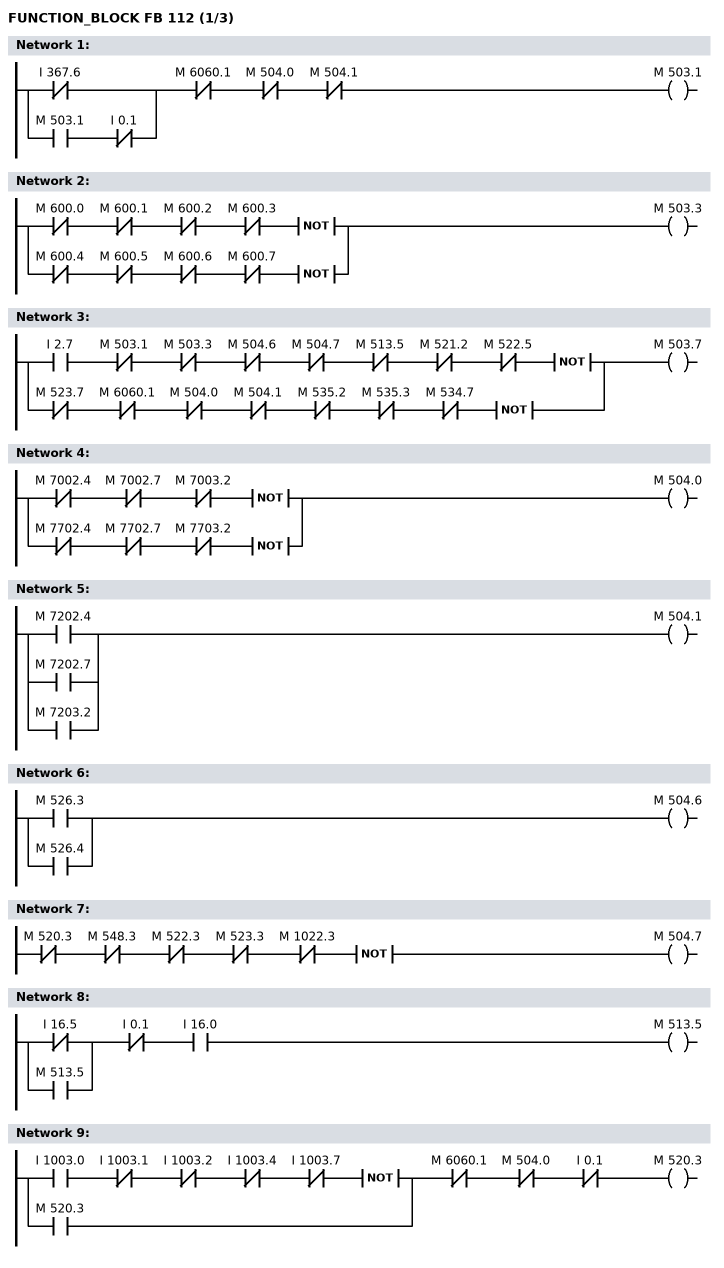

      A(    ;
      ON    I    367.6;
      O     ;
      A     M    503.1;
      AN    I      0.1;
      )     ;
      AN    M   6060.1;
      AN    M    504.0;
      AN    M    504.1;
      =     M    503.1;
NETWORK
TITLE =

      AN    M    600.0;
      AN    M    600.1;
      AN    M    600.2;
      AN    M    600.3;
      NOT   ;
      O(    ;
      AN    M    600.4;
      AN    M    600.5;
      AN    M    600.6;
      AN    M    600.7;
      NOT   ;
      )     ;
      =     M    503.3;
NETWORK
TITLE =

      A     I      2.7;
      AN    M    503.1;
      AN    M    503.3;
      AN    M    504.6;
      AN    M    504.7;
      AN    M    513.5;
      AN    M    521.2;
      AN    M    522.5;
      NOT   ;
      O(    ;
      AN    M    523.7;
      AN    M   6060.1;
      AN    M    504.0;
      AN    M    504.1;
      AN    M    535.2;
      AN    M    535.3;
      AN    M    534.7;
      NOT   ;
      )     ;
      =     M    503.7;
NETWORK
TITLE =

      AN    M   7002.4;
      AN    M   7002.7;
      AN    M   7003.2;
      NOT   ;
      O(    ;
      AN    M   7702.4;
      AN    M   7702.7;
      AN    M   7703.2;
      NOT   ;
      )     ;
      =     M    504.0;
NETWORK
TITLE =

      O     M   7202.4;
      O     M   7202.7;
      O     M   7203.2;
      =     M    504.1;
NETWORK
TITLE =

      O     M    526.3;
      O     M    526.4;
      =     M    504.6;
NETWORK
TITLE =

      AN    M    520.3;
      AN    M    548.3;
      AN    M    522.3;
      AN    M    523.3;
      AN    M   1022.3;
      NOT   ;
      =     M    504.7;
NETWORK
TITLE =

      A(    ;
      ON    I     16.5;
      O     M    513.5;
      )     ;
      AN    I      0.1;
      A     I     16.0;
      =     M    513.5;
NETWORK
TITLE =

      A(    ;
      A     I   1003.0;
      AN    I   1003.1;
      AN    I   1003.2;
      AN    I   1003.4;
      AN    I   1003.7;
      NOT   ;
      O     M    520.3;
      )     ;
      AN    M   6060.1;
      AN    M    504.0;
      AN    I      0.1;
      =     M    520.3;
NETWORK
TITLE =
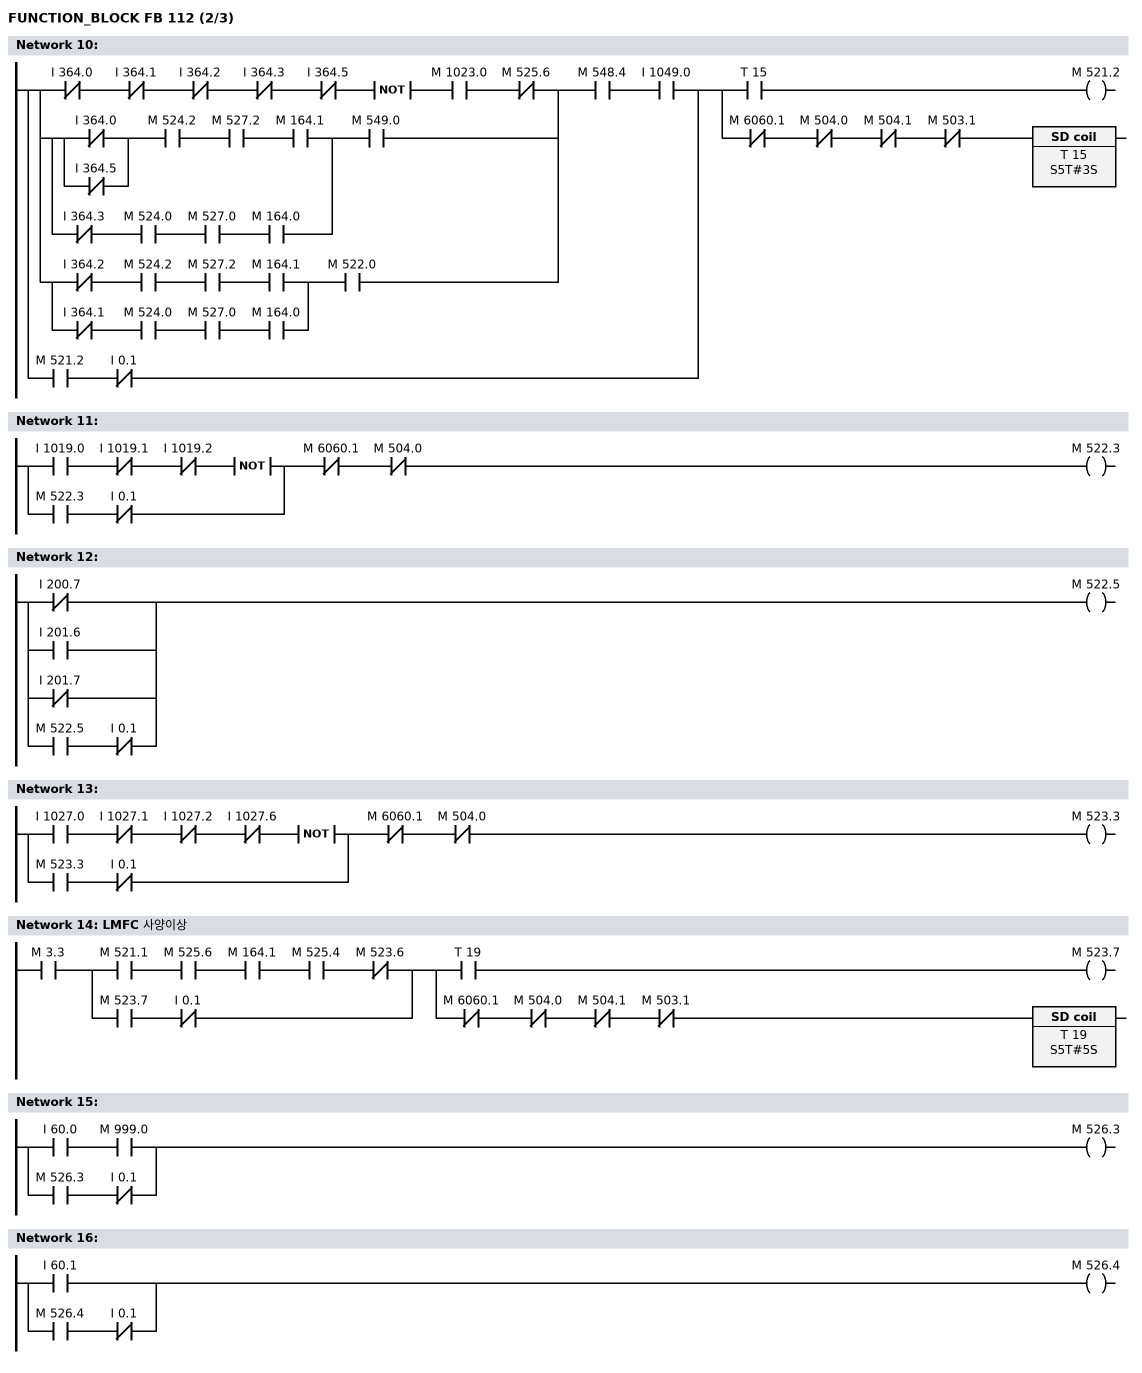

      A(    ;
      AN    I    364.0;
      AN    I    364.1;
      AN    I    364.2;
      AN    I    364.3;
      AN    I    364.5;
      NOT   ;
      A     M   1023.0;
      AN    M    525.6;
      O     ;
      A(    ;
      A(    ;
      ON    I    364.0;
      ON    I    364.5;
      )     ;
      A     M    524.2;
      A     M    527.2;
      A     M    164.1;
      O     ;
      AN    I    364.3;
      A     M    524.0;
      A     M    527.0;
      A     M    164.0;
      )     ;
      A     M    549.0;
      O     ;
      A(    ;
      AN    I    364.2;
      A     M    524.2;
      A     M    527.2;
      A     M    164.1;
      O     ;
      AN    I    364.1;
      A     M    524.0;
      A     M    527.0;
      A     M    164.0;
      )     ;
      A     M    522.0;
      )     ;
      A     M    548.4;
      A     I   1049.0;
      O     ;
      A     M    521.2;
      AN    I      0.1;
      =     L      0.0;
      A     L      0.0;
      A     T     15;
      =     M    521.2;
      A     L      0.0;
      AN    M   6060.1;
      AN    M    504.0;
      AN    M    504.1;
      AN    M    503.1;
      L     S5T#3S;
      SD    T     15;
NETWORK
TITLE =

      A(    ;
      A     I   1019.0;
      AN    I   1019.1;
      AN    I   1019.2;
      NOT   ;
      O     ;
      A     M    522.3;
      AN    I      0.1;
      )     ;
      AN    M   6060.1;
      AN    M    504.0;
      =     M    522.3;
NETWORK
TITLE =

      ON    I    200.7;
      O     I    201.6;
      ON    I    201.7;
      O     ;
      A     M    522.5;
      AN    I      0.1;
      =     M    522.5;
NETWORK
TITLE =

      A(    ;
      A     I   1027.0;
      AN    I   1027.1;
      AN    I   1027.2;
      AN    I   1027.6;
      NOT   ;
      O     ;
      A     M    523.3;
      AN    I      0.1;
      )     ;
      AN    M   6060.1;
      AN    M    504.0;
      =     M    523.3;
NETWORK
TITLE =LMFC 사양이상

      A     M      3.3;
      A(    ;
      A     M    521.1;
      A     M    525.6;
      A     M    164.1;
      A     M    525.4;
      AN    M    523.6;
      O     ;
      A     M    523.7;
      AN    I      0.1;
      )     ;
      =     L      0.0;
      A     L      0.0;
      A     T     19;
      =     M    523.7;
      A     L      0.0;
      AN    M   6060.1;
      AN    M    504.0;
      AN    M    504.1;
      AN    M    503.1;
      L     S5T#5S;
      SD    T     19;
NETWORK
TITLE =

      A     I     60.0;
      A     M    999.0;
      O     ;
      A     M    526.3;
      AN    I      0.1;
      =     M    526.3;
NETWORK
TITLE =

      O     I     60.1;
      O     ;
      A     M    526.4;
      AN    I      0.1;
      =     M    526.4;
NETWORK
TITLE =
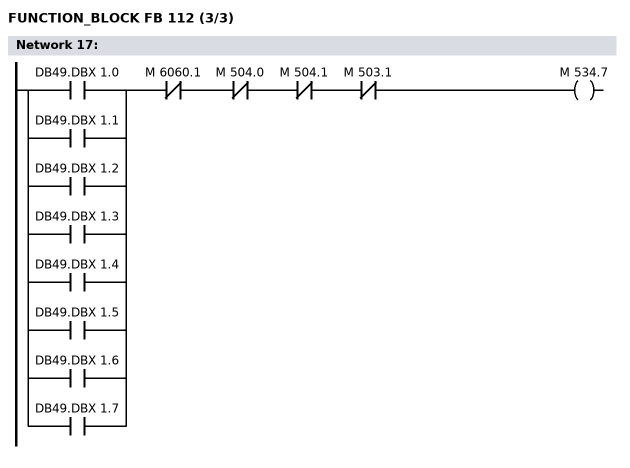

      A(    ;
      O     DB49.DBX    1.0;
      O     DB49.DBX    1.1;
      O     DB49.DBX    1.2;
      O     DB49.DBX    1.3;
      O     DB49.DBX    1.4;
      O     DB49.DBX    1.5;
      O     DB49.DBX    1.6;
      O     DB49.DBX    1.7;
      )     ;
      AN    M   6060.1;
      AN    M    504.0;
      AN    M    504.1;
      AN    M    503.1;
      =     M    534.7;
NETWORK
TITLE =

      A     M      3.3;
      =     L      0.0;
      A     L      0.0;
      A(    ;
      A     M    535.6;
      A(    ;
      ON    M    535.4;
      O     ;
      A     M    535.4;
      A(    ;
      A     I    367.1;
      A     I    367.3;
      O     ;
      AN    I    367.1;
      AN    I    367.3;
      O     ;
      A     M    124.0;
      A     I    367.1;
      AN    I    367.3;
      O     ;
      A     M    124.1;
      AN    I    367.1;
      A     I    367.3;
      )     ;
      )     ;
      A     I   1009.1;
      O     ;
      A     M    535.2;
      AN    I      0.1;
      )     ;
      =     L      0.1;
      A     L      0.1;
      A     T     12;
      =     M    535.2;
      A     L      0.1;
      AN    M   6060.1;
      AN    M    504.0;
      AN    M    504.1;
      AN    M    503.1;
      L     S5T#1S;
      SD    T     12;
      A     L      0.0;
      A(    ;
      A     M    535.7;
      AN    M    535.5;
      A     I   1002.2;
      O     ;
      A     M    535.3;
      AN    I      0.1;
      )     ;
      =     L      0.1;
      A     L      0.1;
      A     T     13;
      =     M    535.3;
      A     L      0.1;
      AN    M   6060.1;
      AN    M    504.0;
      AN    M    504.1;
      AN    M    503.1;
      L     S5T#1S;
      SD    T     13;
NETWORK
TITLE =
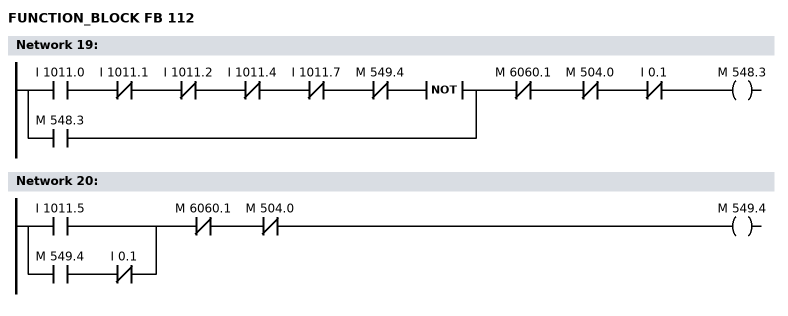

      A(    ;
      A     I   1011.0;
      AN    I   1011.1;
      AN    I   1011.2;
      AN    I   1011.4;
      AN    I   1011.7;
      AN    M    549.4;
      NOT   ;
      O     M    548.3;
      )     ;
      AN    M   6060.1;
      AN    M    504.0;
      AN    I      0.1;
      =     M    548.3;
NETWORK
TITLE =

      A(    ;
      O     I   1011.5;
      O     ;
      A     M    549.4;
      AN    I      0.1;
      )     ;
      AN    M   6060.1;
      AN    M    504.0;
      =     M    549.4;
END_FUNCTION_BLOCK

DATA_BLOCK DB 112
TITLE =
VERSION : 0.0

 FB 112
BEGIN
END_DATA_BLOCK

FUNCTION FC 112 : VOID
TITLE =
VERSION : 0.1

BEGIN
NETWORK
TITLE =

      AN    OV;
      =     L      0.0;
      A     L      0.0;
      A     I    364.6;
      AN    I    364.7;
      A     I    365.0;
      AN    I    365.1;
      =     M    524.0;
      A     L      0.0;
      AN    I    364.6;
      A     I    364.7;
      AN    I    365.0;
      A     I    365.1;
      =     M    524.1;
NETWORK
TITLE =

      AN    OV;
      =     L      0.0;
      A     L      0.0;
      A     I    365.2;
      AN    I    365.3;
      A     I    365.4;
      AN    I    365.5;
      =     M    524.2;
      A     L      0.0;
      AN    I    365.2;
      A     I    365.3;
      AN    I    365.4;
      A     I    365.5;
      =     M    524.3;
NETWORK
TITLE =

      AN    OV;
      =     L      0.0;
      A     L      0.0;
      A     I    366.0;
      AN    I    366.1;
      A     I    366.2;
      AN    I    366.3;
      =     M    527.0;
      A     L      0.0;
      AN    I    366.0;
      A     I    366.1;
      AN    I    366.2;
      A     I    366.3;
      =     M    527.1;
NETWORK
TITLE =

      AN    OV;
      =     L      0.0;
      A     L      0.0;
      A     I    366.4;
      AN    I    366.5;
      A     I    366.6;
      AN    I    366.7;
      =     M    527.2;
      A     L      0.0;
      AN    I    366.4;
      A     I    366.5;
      AN    I    366.6;
      A     I    366.7;
      =     M    527.3;
NETWORK
TITLE =
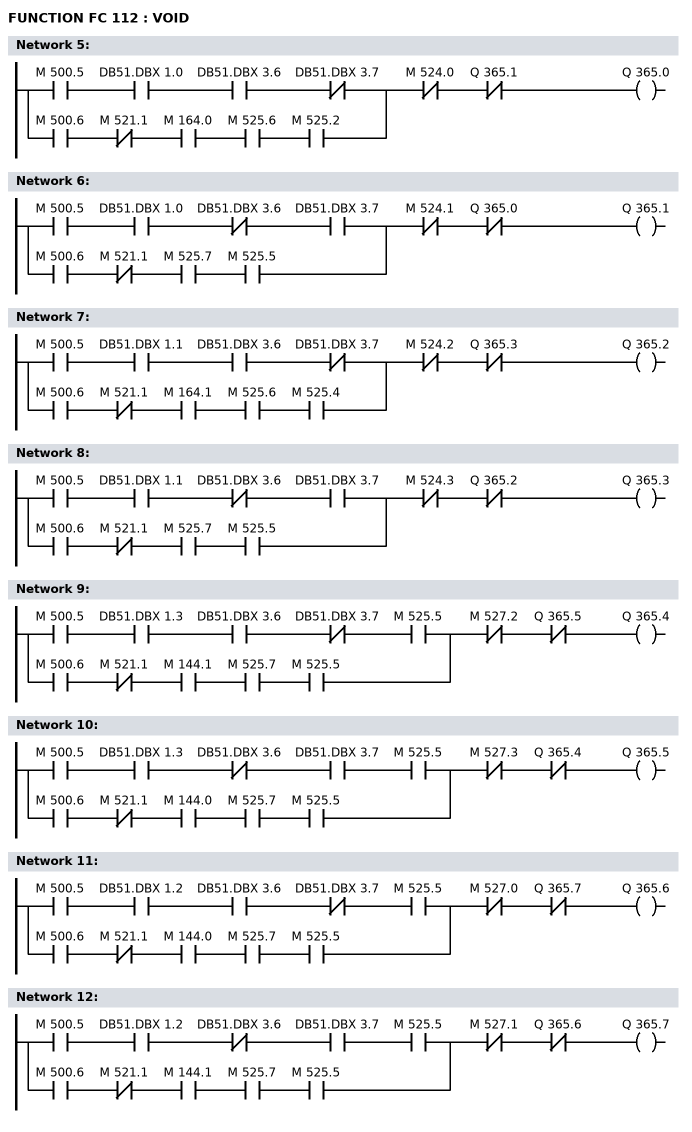

      A(    ;
      A     M    500.5;
      A     DB51.DBX    1.0;
      A     DB51.DBX    3.6;
      AN    DB51.DBX    3.7;
      O     ;
      A     M    500.6;
      AN    M    521.1;
      A     M    164.0;
      A     M    525.6;
      A     M    525.2;
      )     ;
      AN    M    524.0;
      AN    Q    365.1;
      =     Q    365.0;
NETWORK
TITLE =

      A(    ;
      A     M    500.5;
      A     DB51.DBX    1.0;
      AN    DB51.DBX    3.6;
      A     DB51.DBX    3.7;
      O     ;
      A     M    500.6;
      AN    M    521.1;
      A     M    525.7;
      A     M    525.5;
      )     ;
      AN    M    524.1;
      AN    Q    365.0;
      =     Q    365.1;
NETWORK
TITLE =

      A(    ;
      A     M    500.5;
      A     DB51.DBX    1.1;
      A     DB51.DBX    3.6;
      AN    DB51.DBX    3.7;
      O     ;
      A     M    500.6;
      AN    M    521.1;
      A     M    164.1;
      A     M    525.6;
      A     M    525.4;
      )     ;
      AN    M    524.2;
      AN    Q    365.3;
      =     Q    365.2;
NETWORK
TITLE =

      A(    ;
      A     M    500.5;
      A     DB51.DBX    1.1;
      AN    DB51.DBX    3.6;
      A     DB51.DBX    3.7;
      O     ;
      A     M    500.6;
      AN    M    521.1;
      A     M    525.7;
      A     M    525.5;
      )     ;
      AN    M    524.3;
      AN    Q    365.2;
      =     Q    365.3;
NETWORK
TITLE =

      A(    ;
      A     M    500.5;
      A     DB51.DBX    1.3;
      A     DB51.DBX    3.6;
      AN    DB51.DBX    3.7;
      A     M    525.5;
      O     ;
      A     M    500.6;
      AN    M    521.1;
      A     M    144.1;
      A     M    525.7;
      A     M    525.5;
      )     ;
      AN    M    527.2;
      AN    Q    365.5;
      =     Q    365.4;
NETWORK
TITLE =

      A(    ;
      A     M    500.5;
      A     DB51.DBX    1.3;
      AN    DB51.DBX    3.6;
      A     DB51.DBX    3.7;
      A     M    525.5;
      O     ;
      A     M    500.6;
      AN    M    521.1;
      A     M    144.0;
      A     M    525.7;
      A     M    525.5;
      )     ;
      AN    M    527.3;
      AN    Q    365.4;
      =     Q    365.5;
NETWORK
TITLE =

      A(    ;
      A     M    500.5;
      A     DB51.DBX    1.2;
      A     DB51.DBX    3.6;
      AN    DB51.DBX    3.7;
      A     M    525.5;
      O     ;
      A     M    500.6;
      AN    M    521.1;
      A     M    144.0;
      A     M    525.7;
      A     M    525.5;
      )     ;
      AN    M    527.0;
      AN    Q    365.7;
      =     Q    365.6;
NETWORK
TITLE =

      A(    ;
      A     M    500.5;
      A     DB51.DBX    1.2;
      AN    DB51.DBX    3.6;
      A     DB51.DBX    3.7;
      A     M    525.5;
      O     ;
      A     M    500.6;
      AN    M    521.1;
      A     M    144.1;
      A     M    525.7;
      A     M    525.5;
      )     ;
      AN    M    527.1;
      AN    Q    365.6;
      =     Q    365.7;
END_FUNCTION

FUNCTION FC 113 : VOID
TITLE =
VERSION : 0.1

BEGIN
NETWORK
TITLE =

      A     I   1000.0;
      JNB   _001;
      L     0;
      T     MW   590;
_001: NOP   0;
NETWORK
TITLE =

      AN    OV;
      =     L      0.0;
      A     L      0.0;
      A     M    104.1;
      =     L      0.1;
      A     L      0.1;
      A     T    363;
      A(    ;
      L     1;
      L     DB59.DBW   34;
      ==I   ;
      )     ;
      A(    ;
      L     1;
      L     DB59.DBW   30;
      ==I   ;
      )     ;
      A     M    550.3;
      JNB   _002;
      L     23;
      T     MB   591;
_002: NOP   0;
      A     L      0.1;
      A     T    364;
      A(    ;
      L     1;
      L     DB59.DBW   44;
      ==I   ;
      )     ;
      A(    ;
      L     1;
      L     DB59.DBW   40;
      ==I   ;
      )     ;
      A     M    550.4;
      JNB   _003;
      L     24;
      T     MB   591;
_003: NOP   0;
      A     L      0.1;
      A     T    365;
      A(    ;
      L     1;
      L     DB59.DBW   54;
      ==I   ;
      )     ;
      A(    ;
      L     1;
      L     DB59.DBW   50;
      ==I   ;
      )     ;
      A     M    550.5;
      JNB   _004;
      L     25;
      T     MB   591;
_004: NOP   0;
      A     L      0.1;
      A     T    366;
      A(    ;
      L     1;
      L     DB59.DBW   64;
      ==I   ;
      )     ;
      A(    ;
      L     1;
      L     DB59.DBW   60;
      ==I   ;
      )     ;
      A     M    550.6;
      JNB   _005;
      L     26;
      T     MB   591;
_005: NOP   0;
      A     L      0.0;
      A     M    104.0;
      =     L      0.1;
      A     L      0.1;
      A     T    363;
      A(    ;
      L     1;
      L     DB59.DBW   34;
      ==I   ;
      )     ;
      A(    ;
      L     2;
      L     DB59.DBW   30;
      ==I   ;
      )     ;
      A     M    554.3;
      JNB   _006;
      L     3;
      T     MB   591;
_006: NOP   0;
      A     L      0.1;
      A     T    364;
      A(    ;
      L     1;
      L     DB59.DBW   44;
      ==I   ;
      )     ;
      A(    ;
      L     2;
      L     DB59.DBW   40;
      ==I   ;
      )     ;
      A     M    554.4;
      JNB   _007;
      L     4;
      T     MB   591;
_007: NOP   0;
      A     L      0.1;
      A     T    365;
      A(    ;
      L     1;
      L     DB59.DBW   54;
      ==I   ;
      )     ;
      A(    ;
      L     2;
      L     DB59.DBW   50;
      ==I   ;
      )     ;
      A     M    554.5;
      JNB   _008;
      L     5;
      T     MB   591;
_008: NOP   0;
      A     L      0.1;
      A     T    366;
      A(    ;
      L     1;
      L     DB59.DBW   64;
      ==I   ;
      )     ;
      A(    ;
      L     2;
      L     DB59.DBW   60;
      ==I   ;
      )     ;
      A     M    554.6;
      JNB   _009;
      L     6;
      T     MB   591;
_009: NOP   0;
NETWORK
TITLE =

      AN    OV;
      =     L      0.0;
      A     L      0.0;
      A     M    104.1;
      =     L      0.1;
      A     L      0.1;
      A     T    369;
      A(    ;
      L     1;
      L     DB59.DBW   94;
      ==I   ;
      )     ;
      A(    ;
      L     1;
      L     DB59.DBW   90;
      ==I   ;
      )     ;
      A     M    551.1;
      JNB   _00a;
      L     29;
      T     MB   591;
_00a: NOP   0;
      A     L      0.1;
      A     T    370;
      A(    ;
      L     1;
      L     DB59.DBW  104;
      ==I   ;
      )     ;
      A(    ;
      L     1;
      L     DB59.DBW  100;
      ==I   ;
      )     ;
      A     M    551.2;
      JNB   _00b;
      L     30;
      T     MB   591;
_00b: NOP   0;
      A     L      0.1;
      A     T    371;
      A(    ;
      L     1;
      L     DB59.DBW  114;
      ==I   ;
      )     ;
      A(    ;
      L     1;
      L     DB59.DBW  110;
      ==I   ;
      )     ;
      A     M    551.3;
      JNB   _00c;
      L     31;
      T     MB   591;
_00c: NOP   0;
      A     L      0.1;
      A     T    372;
      A(    ;
      L     1;
      L     DB59.DBW  124;
      ==I   ;
      )     ;
      A(    ;
      L     1;
      L     DB59.DBW  120;
      ==I   ;
      )     ;
      A     M    551.4;
      JNB   _00d;
      L     32;
      T     MB   591;
_00d: NOP   0;
      A     L      0.0;
      A     M    104.0;
      =     L      0.1;
      A     L      0.1;
      A     T    369;
      A(    ;
      L     1;
      L     DB59.DBW   94;
      ==I   ;
      )     ;
      A(    ;
      L     2;
      L     DB59.DBW   90;
      ==I   ;
      )     ;
      A     M    555.1;
      JNB   _00e;
      L     9;
      T     MB   591;
_00e: NOP   0;
      A     L      0.1;
      A     T    370;
      A(    ;
      L     1;
      L     DB59.DBW  104;
      ==I   ;
      )     ;
      A(    ;
      L     2;
      L     DB59.DBW  100;
      ==I   ;
      )     ;
      A     M    555.2;
      JNB   _00f;
      L     10;
      T     MB   591;
_00f: NOP   0;
      A     L      0.1;
      A     T    371;
      A(    ;
      L     1;
      L     DB59.DBW  114;
      ==I   ;
      )     ;
      A(    ;
      L     2;
      L     DB59.DBW  110;
      ==I   ;
      )     ;
      A     M    555.3;
      JNB   _010;
      L     11;
      T     MB   591;
_010: NOP   0;
      A     L      0.1;
      A     T    372;
      A(    ;
      L     1;
      L     DB59.DBW  124;
      ==I   ;
      )     ;
      A(    ;
      L     2;
      L     DB59.DBW  120;
      ==I   ;
      )     ;
      A     M    555.4;
      JNB   _011;
      L     12;
      T     MB   591;
_011: NOP   0;
NETWORK
TITLE =
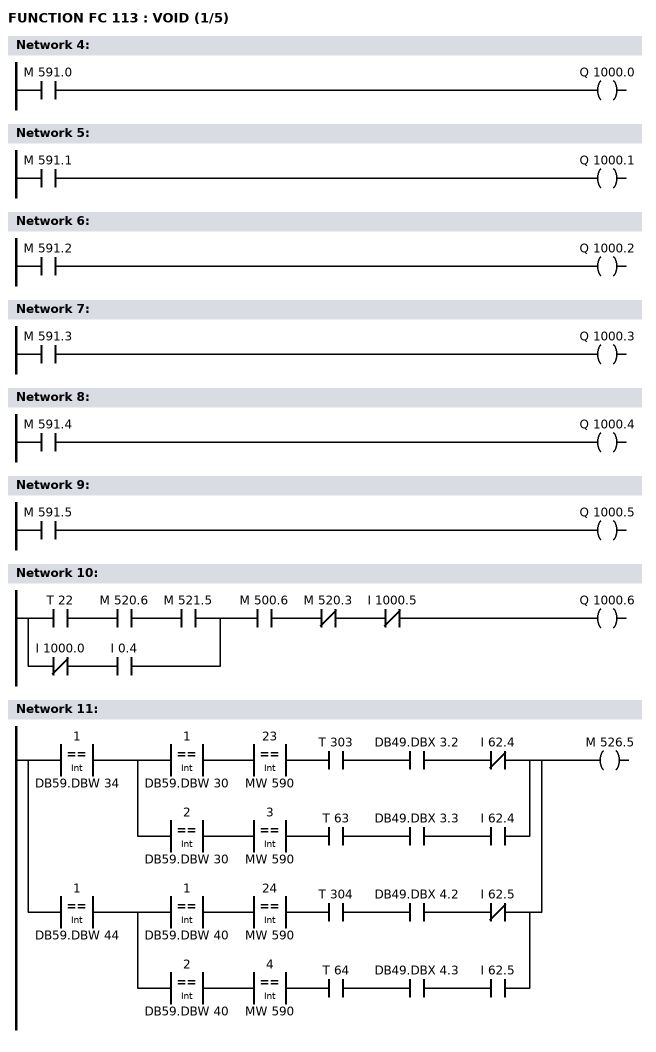

      A     M    591.0;
      =     Q   1000.0;
NETWORK
TITLE =

      A     M    591.1;
      =     Q   1000.1;
NETWORK
TITLE =

      A     M    591.2;
      =     Q   1000.2;
NETWORK
TITLE =

      A     M    591.3;
      =     Q   1000.3;
NETWORK
TITLE =

      A     M    591.4;
      =     Q   1000.4;
NETWORK
TITLE =

      A     M    591.5;
      =     Q   1000.5;
NETWORK
TITLE =

      A(    ;
      A     T     22;
      A     M    520.6;
      A     M    521.5;
      O     ;
      AN    I   1000.0;
      A     I      0.4;
      )     ;
      A     M    500.6;
      AN    M    520.3;
      AN    I   1000.5;
      =     Q   1000.6;
NETWORK
TITLE =

      A(    ;
      L     1;
      L     DB59.DBW   34;
      ==I   ;
      )     ;
      A(    ;
      A(    ;
      L     1;
      L     DB59.DBW   30;
      ==I   ;
      )     ;
      A(    ;
      L     23;
      L     MW   590;
      ==I   ;
      )     ;
      A     T    303;
      A     DB49.DBX    3.2;
      AN    I     62.4;
      O     ;
      A(    ;
      L     2;
      L     DB59.DBW   30;
      ==I   ;
      )     ;
      A(    ;
      L     3;
      L     MW   590;
      ==I   ;
      )     ;
      A     T     63;
      A     DB49.DBX    3.3;
      A     I     62.4;
      )     ;
      O     ;
      A(    ;
      L     1;
      L     DB59.DBW   44;
      ==I   ;
      )     ;
      A(    ;
      A(    ;
      L     1;
      L     DB59.DBW   40;
      ==I   ;
      )     ;
      A(    ;
      L     24;
      L     MW   590;
      ==I   ;
      )     ;
      A     T    304;
      A     DB49.DBX    4.2;
      AN    I     62.5;
      O     ;
      A(    ;
      L     2;
      L     DB59.DBW   40;
      ==I   ;
      )     ;
      A(    ;
      L     4;
      L     MW   590;
      ==I   ;
      )     ;
      A     T     64;
      A     DB49.DBX    4.3;
      A     I     62.5;
      )     ;
      =     M    526.5;
NETWORK
TITLE =
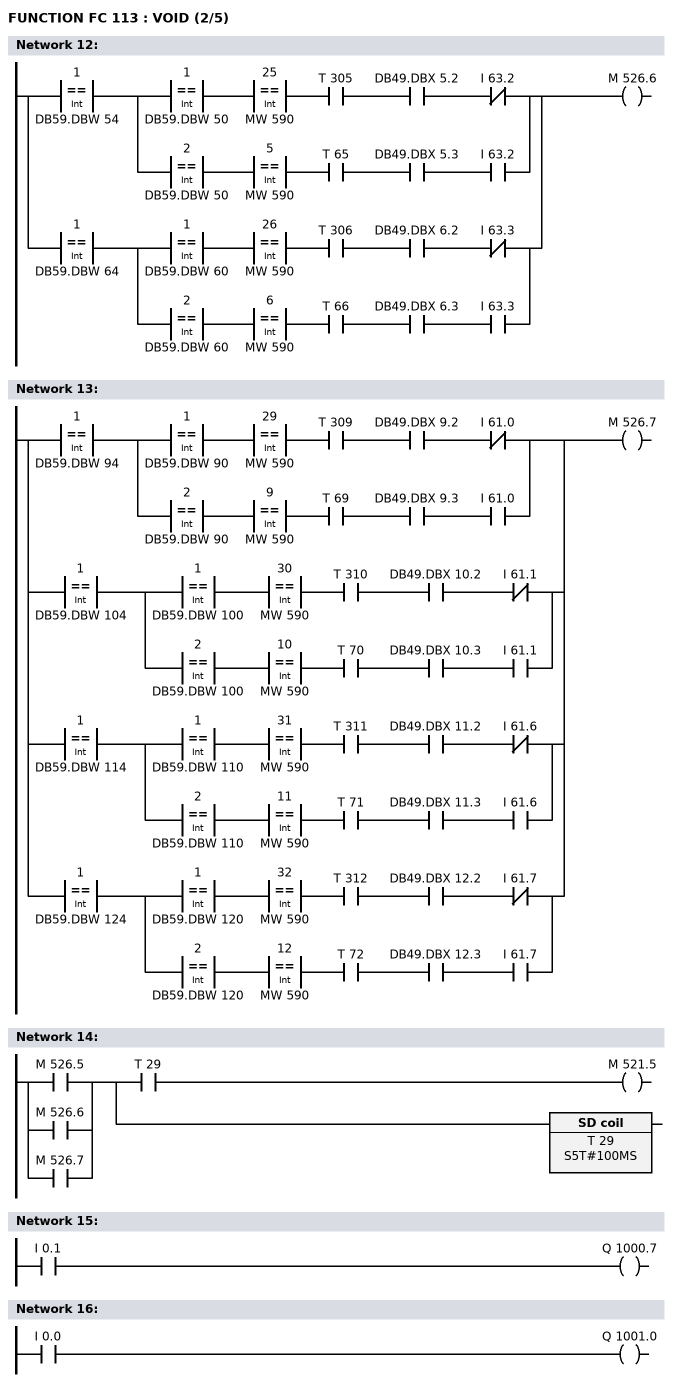

      A(    ;
      L     1;
      L     DB59.DBW   54;
      ==I   ;
      )     ;
      A(    ;
      A(    ;
      L     1;
      L     DB59.DBW   50;
      ==I   ;
      )     ;
      A(    ;
      L     25;
      L     MW   590;
      ==I   ;
      )     ;
      A     T    305;
      A     DB49.DBX    5.2;
      AN    I     63.2;
      O     ;
      A(    ;
      L     2;
      L     DB59.DBW   50;
      ==I   ;
      )     ;
      A(    ;
      L     5;
      L     MW   590;
      ==I   ;
      )     ;
      A     T     65;
      A     DB49.DBX    5.3;
      A     I     63.2;
      )     ;
      O     ;
      A(    ;
      L     1;
      L     DB59.DBW   64;
      ==I   ;
      )     ;
      A(    ;
      A(    ;
      L     1;
      L     DB59.DBW   60;
      ==I   ;
      )     ;
      A(    ;
      L     26;
      L     MW   590;
      ==I   ;
      )     ;
      A     T    306;
      A     DB49.DBX    6.2;
      AN    I     63.3;
      O     ;
      A(    ;
      L     2;
      L     DB59.DBW   60;
      ==I   ;
      )     ;
      A(    ;
      L     6;
      L     MW   590;
      ==I   ;
      )     ;
      A     T     66;
      A     DB49.DBX    6.3;
      A     I     63.3;
      )     ;
      =     M    526.6;
NETWORK
TITLE =

      A(    ;
      L     1;
      L     DB59.DBW   94;
      ==I   ;
      )     ;
      A(    ;
      A(    ;
      L     1;
      L     DB59.DBW   90;
      ==I   ;
      )     ;
      A(    ;
      L     29;
      L     MW   590;
      ==I   ;
      )     ;
      A     T    309;
      A     DB49.DBX    9.2;
      AN    I     61.0;
      O     ;
      A(    ;
      L     2;
      L     DB59.DBW   90;
      ==I   ;
      )     ;
      A(    ;
      L     9;
      L     MW   590;
      ==I   ;
      )     ;
      A     T     69;
      A     DB49.DBX    9.3;
      A     I     61.0;
      )     ;
      O     ;
      A(    ;
      L     1;
      L     DB59.DBW  104;
      ==I   ;
      )     ;
      A(    ;
      A(    ;
      L     1;
      L     DB59.DBW  100;
      ==I   ;
      )     ;
      A(    ;
      L     30;
      L     MW   590;
      ==I   ;
      )     ;
      A     T    310;
      A     DB49.DBX   10.2;
      AN    I     61.1;
      O     ;
      A(    ;
      L     2;
      L     DB59.DBW  100;
      ==I   ;
      )     ;
      A(    ;
      L     10;
      L     MW   590;
      ==I   ;
      )     ;
      A     T     70;
      A     DB49.DBX   10.3;
      A     I     61.1;
      )     ;
      O     ;
      A(    ;
      L     1;
      L     DB59.DBW  114;
      ==I   ;
      )     ;
      A(    ;
      A(    ;
      L     1;
      L     DB59.DBW  110;
      ==I   ;
      )     ;
      A(    ;
      L     31;
      L     MW   590;
      ==I   ;
      )     ;
      A     T    311;
      A     DB49.DBX   11.2;
      AN    I     61.6;
      O     ;
      A(    ;
      L     2;
      L     DB59.DBW  110;
      ==I   ;
      )     ;
      A(    ;
      L     11;
      L     MW   590;
      ==I   ;
      )     ;
      A     T     71;
      A     DB49.DBX   11.3;
      A     I     61.6;
      )     ;
      O     ;
      A(    ;
      L     1;
      L     DB59.DBW  124;
      ==I   ;
      )     ;
      A(    ;
      A(    ;
      L     1;
      L     DB59.DBW  120;
      ==I   ;
      )     ;
      A(    ;
      L     32;
      L     MW   590;
      ==I   ;
      )     ;
      A     T    312;
      A     DB49.DBX   12.2;
      AN    I     61.7;
      O     ;
      A(    ;
      L     2;
      L     DB59.DBW  120;
      ==I   ;
      )     ;
      A(    ;
      L     12;
      L     MW   590;
      ==I   ;
      )     ;
      A     T     72;
      A     DB49.DBX   12.3;
      A     I     61.7;
      )     ;
      =     M    526.7;
NETWORK
TITLE =

      O     M    526.5;
      O     M    526.6;
      O     M    526.7;
      =     L      0.0;
      A     L      0.0;
      A     T     29;
      =     M    521.5;
      A     L      0.0;
      BLD   102;
      L     S5T#100MS;
      SD    T     29;
NETWORK
TITLE =

      A     I      0.1;
      =     Q   1000.7;
NETWORK
TITLE =

      A     I      0.0;
      =     Q   1001.0;
NETWORK
TITLE =
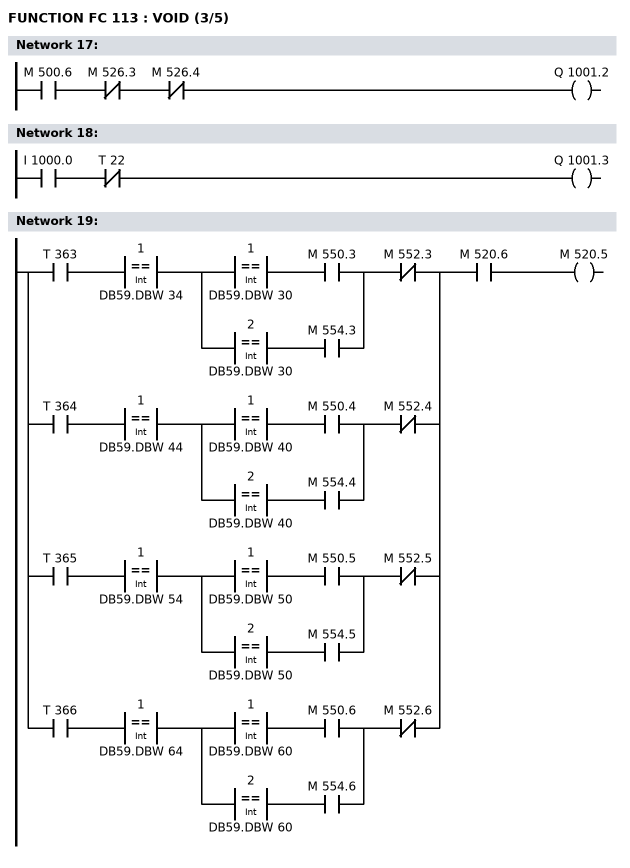

      A     M    500.6;
      AN    M    526.3;
      AN    M    526.4;
      =     Q   1001.2;
NETWORK
TITLE =

      A     I   1000.0;
      AN    T     22;
      =     Q   1001.3;
NETWORK
TITLE =

      A(    ;
      A     T    363;
      A(    ;
      L     1;
      L     DB59.DBW   34;
      ==I   ;
      )     ;
      A(    ;
      A(    ;
      L     1;
      L     DB59.DBW   30;
      ==I   ;
      )     ;
      A     M    550.3;
      O     ;
      A(    ;
      L     2;
      L     DB59.DBW   30;
      ==I   ;
      )     ;
      A     M    554.3;
      )     ;
      AN    M    552.3;
      O     ;
      A     T    364;
      A(    ;
      L     1;
      L     DB59.DBW   44;
      ==I   ;
      )     ;
      A(    ;
      A(    ;
      L     1;
      L     DB59.DBW   40;
      ==I   ;
      )     ;
      A     M    550.4;
      O     ;
      A(    ;
      L     2;
      L     DB59.DBW   40;
      ==I   ;
      )     ;
      A     M    554.4;
      )     ;
      AN    M    552.4;
      O     ;
      A     T    365;
      A(    ;
      L     1;
      L     DB59.DBW   54;
      ==I   ;
      )     ;
      A(    ;
      A(    ;
      L     1;
      L     DB59.DBW   50;
      ==I   ;
      )     ;
      A     M    550.5;
      O     ;
      A(    ;
      L     2;
      L     DB59.DBW   50;
      ==I   ;
      )     ;
      A     M    554.5;
      )     ;
      AN    M    552.5;
      O     ;
      A     T    366;
      A(    ;
      L     1;
      L     DB59.DBW   64;
      ==I   ;
      )     ;
      A(    ;
      A(    ;
      L     1;
      L     DB59.DBW   60;
      ==I   ;
      )     ;
      A     M    550.6;
      O     ;
      A(    ;
      L     2;
      L     DB59.DBW   60;
      ==I   ;
      )     ;
      A     M    554.6;
      )     ;
      AN    M    552.6;
      )     ;
      A     M    520.6;
      =     M    520.5;
NETWORK
TITLE =
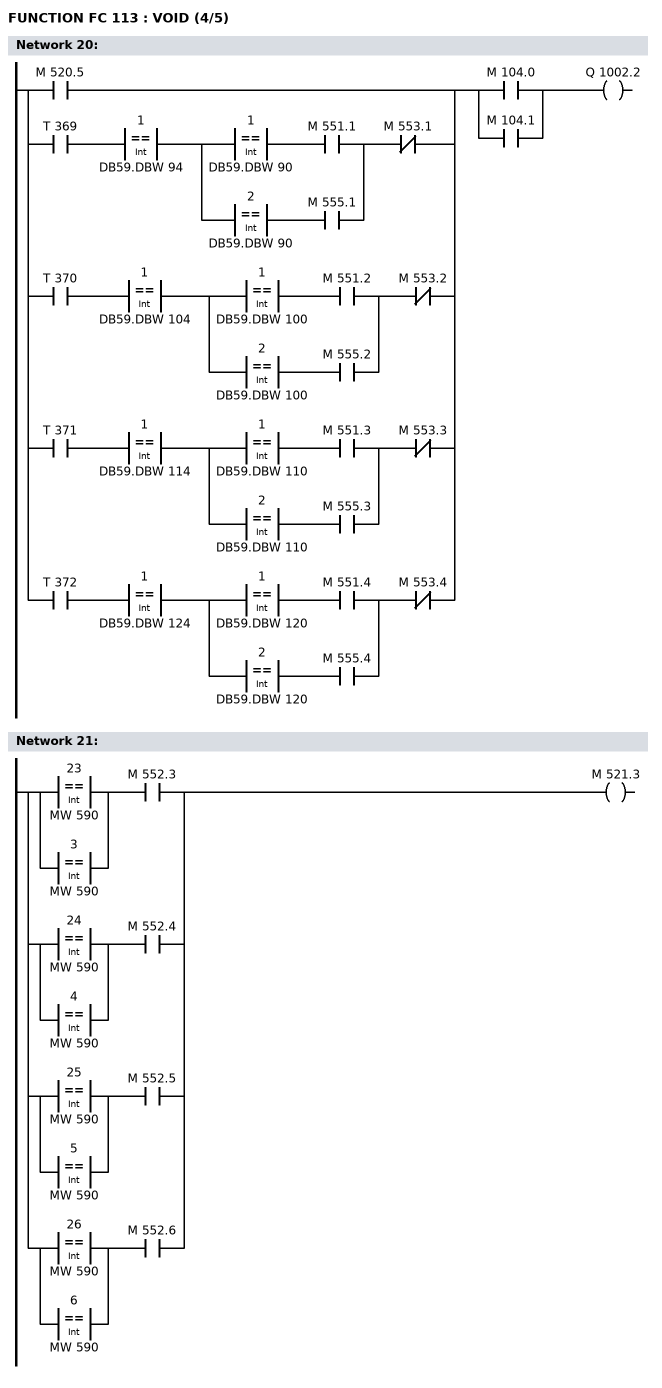

      A(    ;
      O     M    520.5;
      O     ;
      A     T    369;
      A(    ;
      L     1;
      L     DB59.DBW   94;
      ==I   ;
      )     ;
      A(    ;
      A(    ;
      L     1;
      L     DB59.DBW   90;
      ==I   ;
      )     ;
      A     M    551.1;
      O     ;
      A(    ;
      L     2;
      L     DB59.DBW   90;
      ==I   ;
      )     ;
      A     M    555.1;
      )     ;
      AN    M    553.1;
      O     ;
      A     T    370;
      A(    ;
      L     1;
      L     DB59.DBW  104;
      ==I   ;
      )     ;
      A(    ;
      A(    ;
      L     1;
      L     DB59.DBW  100;
      ==I   ;
      )     ;
      A     M    551.2;
      O     ;
      A(    ;
      L     2;
      L     DB59.DBW  100;
      ==I   ;
      )     ;
      A     M    555.2;
      )     ;
      AN    M    553.2;
      O     ;
      A     T    371;
      A(    ;
      L     1;
      L     DB59.DBW  114;
      ==I   ;
      )     ;
      A(    ;
      A(    ;
      L     1;
      L     DB59.DBW  110;
      ==I   ;
      )     ;
      A     M    551.3;
      O     ;
      A(    ;
      L     2;
      L     DB59.DBW  110;
      ==I   ;
      )     ;
      A     M    555.3;
      )     ;
      AN    M    553.3;
      O     ;
      A     T    372;
      A(    ;
      L     1;
      L     DB59.DBW  124;
      ==I   ;
      )     ;
      A(    ;
      A(    ;
      L     1;
      L     DB59.DBW  120;
      ==I   ;
      )     ;
      A     M    551.4;
      O     ;
      A(    ;
      L     2;
      L     DB59.DBW  120;
      ==I   ;
      )     ;
      A     M    555.4;
      )     ;
      AN    M    553.4;
      )     ;
      A(    ;
      O     M    104.0;
      O     M    104.1;
      )     ;
      =     Q   1002.2;
NETWORK
TITLE =

      A(    ;
      O(    ;
      L     23;
      L     MW   590;
      ==I   ;
      )     ;
      O(    ;
      L     3;
      L     MW   590;
      ==I   ;
      )     ;
      )     ;
      A     M    552.3;
      O     ;
      A(    ;
      O(    ;
      L     24;
      L     MW   590;
      ==I   ;
      )     ;
      O(    ;
      L     4;
      L     MW   590;
      ==I   ;
      )     ;
      )     ;
      A     M    552.4;
      O     ;
      A(    ;
      O(    ;
      L     25;
      L     MW   590;
      ==I   ;
      )     ;
      O(    ;
      L     5;
      L     MW   590;
      ==I   ;
      )     ;
      )     ;
      A     M    552.5;
      O     ;
      A(    ;
      O(    ;
      L     26;
      L     MW   590;
      ==I   ;
      )     ;
      O(    ;
      L     6;
      L     MW   590;
      ==I   ;
      )     ;
      )     ;
      A     M    552.6;
      =     M    521.3;
NETWORK
TITLE =
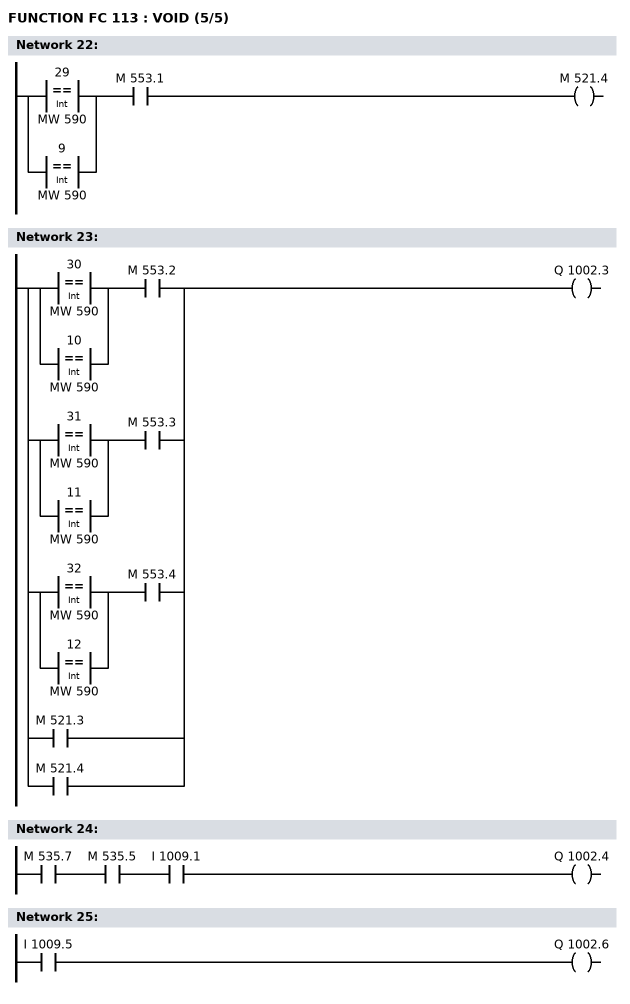

      A(    ;
      O(    ;
      L     29;
      L     MW   590;
      ==I   ;
      )     ;
      O(    ;
      L     9;
      L     MW   590;
      ==I   ;
      )     ;
      )     ;
      A     M    553.1;
      =     M    521.4;
NETWORK
TITLE =

      A(    ;
      O(    ;
      L     30;
      L     MW   590;
      ==I   ;
      )     ;
      O(    ;
      L     10;
      L     MW   590;
      ==I   ;
      )     ;
      )     ;
      A     M    553.2;
      O     ;
      A(    ;
      O(    ;
      L     31;
      L     MW   590;
      ==I   ;
      )     ;
      O(    ;
      L     11;
      L     MW   590;
      ==I   ;
      )     ;
      )     ;
      A     M    553.3;
      O     ;
      A(    ;
      O(    ;
      L     32;
      L     MW   590;
      ==I   ;
      )     ;
      O(    ;
      L     12;
      L     MW   590;
      ==I   ;
      )     ;
      )     ;
      A     M    553.4;
      O     M    521.3;
      O     M    521.4;
      =     Q   1002.3;
NETWORK
TITLE =

      A     M    535.7;
      A     M    535.5;
      A     I   1009.1;
      =     Q   1002.4;
NETWORK
TITLE =

      A     I   1009.5;
      =     Q   1002.6;
END_FUNCTION

FUNCTION FC 114 : VOID
TITLE =
VERSION : 0.1

BEGIN
NETWORK
TITLE =

      A     I   1008.0;
      JNB   _001;
      L     0;
      T     MB   593;
_001: NOP   0;
NETWORK
TITLE =

      AN    OV;
      =     L      0.0;
      A     L      0.0;
      A     M    124.1;
      =     L      0.1;
      A     L      0.1;
      AN    M    127.7;
      A     I   1008.0;
      JNB   _002;
      L     11;
      T     MB   593;
_002: NOP   0;
      A     L      0.1;
      A     M    127.7;
      A     I   1008.0;
      JNB   _003;
      L     19;
      T     MB   593;
_003: NOP   0;
      A     L      0.0;
      A     M    124.0;
      A     I   1008.0;
      JNB   _004;
      L     1;
      T     MB   593;
_004: NOP   0;
NETWORK
TITLE =
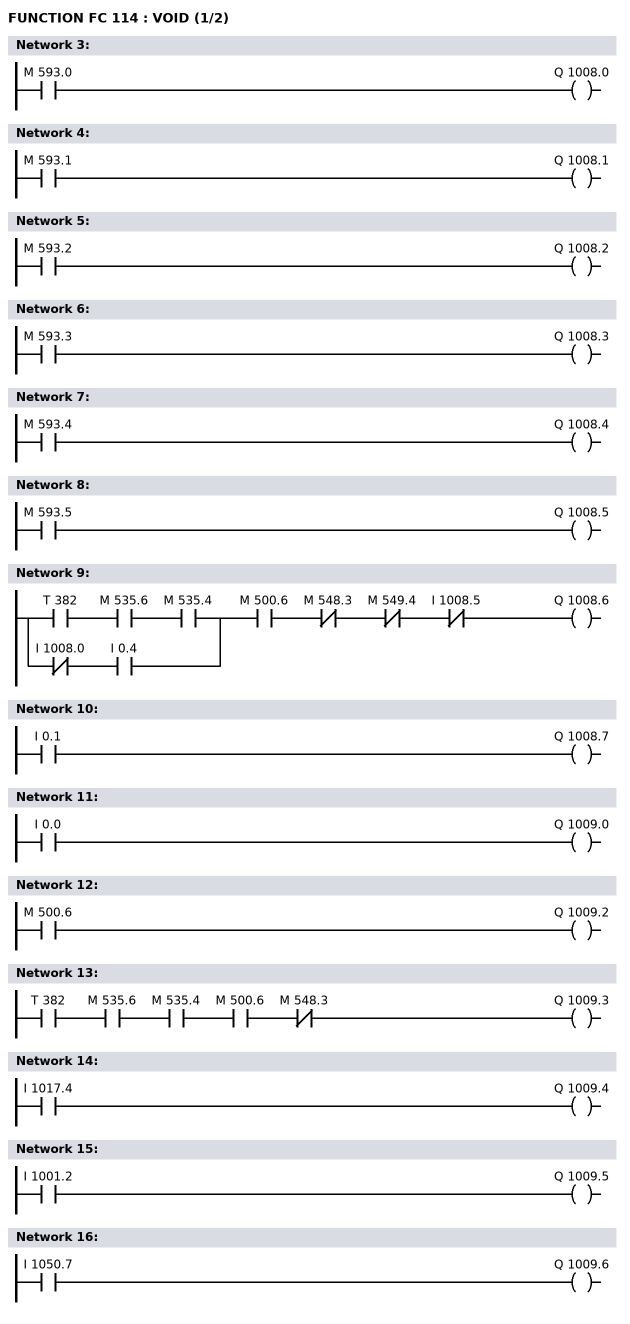

      A     M    593.0;
      =     Q   1008.0;
NETWORK
TITLE =

      A     M    593.1;
      =     Q   1008.1;
NETWORK
TITLE =

      A     M    593.2;
      =     Q   1008.2;
NETWORK
TITLE =

      A     M    593.3;
      =     Q   1008.3;
NETWORK
TITLE =

      A     M    593.4;
      =     Q   1008.4;
NETWORK
TITLE =

      A     M    593.5;
      =     Q   1008.5;
NETWORK
TITLE =

      A(    ;
      A     T    382;
      A     M    535.6;
      A     M    535.4;
      O     ;
      AN    I   1008.0;
      A     I      0.4;
      )     ;
      A     M    500.6;
      AN    M    548.3;
      AN    M    549.4;
      AN    I   1008.5;
      =     Q   1008.6;
NETWORK
TITLE =

      A     I      0.1;
      =     Q   1008.7;
NETWORK
TITLE =

      A     I      0.0;
      =     Q   1009.0;
NETWORK
TITLE =

      A     M    500.6;
      =     Q   1009.2;
NETWORK
TITLE =

      A     T    382;
      A     M    535.6;
      A     M    535.4;
      A     M    500.6;
      AN    M    548.3;
      =     Q   1009.3;
NETWORK
TITLE =

      A     I   1017.4;
      =     Q   1009.4;
NETWORK
TITLE =

      A     I   1001.2;
      =     Q   1009.5;
NETWORK
TITLE =

      A     I   1050.7;
      =     Q   1009.6;
NETWORK
TITLE =
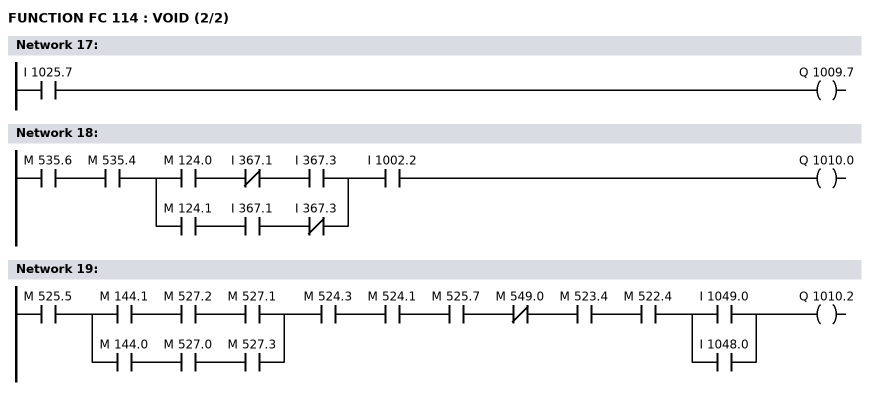

      A     I   1025.7;
      =     Q   1009.7;
NETWORK
TITLE =

      A     M    535.6;
      A     M    535.4;
      A(    ;
      A     M    124.0;
      AN    I    367.1;
      A     I    367.3;
      O     ;
      A     M    124.1;
      A     I    367.1;
      AN    I    367.3;
      )     ;
      A     I   1002.2;
      =     Q   1010.0;
NETWORK
TITLE =

      A     M    525.5;
      A(    ;
      A     M    144.1;
      A     M    527.2;
      A     M    527.1;
      O     ;
      A     M    144.0;
      A     M    527.0;
      A     M    527.3;
      )     ;
      A     M    524.3;
      A     M    524.1;
      A     M    525.7;
      AN    M    549.0;
      A     M    523.4;
      A     M    522.4;
      A(    ;
      O     I   1049.0;
      O     I   1048.0;
      )     ;
      =     Q   1010.2;
END_FUNCTION

FUNCTION FC 115 : VOID
TITLE =
VERSION : 0.1

BEGIN
NETWORK
TITLE =
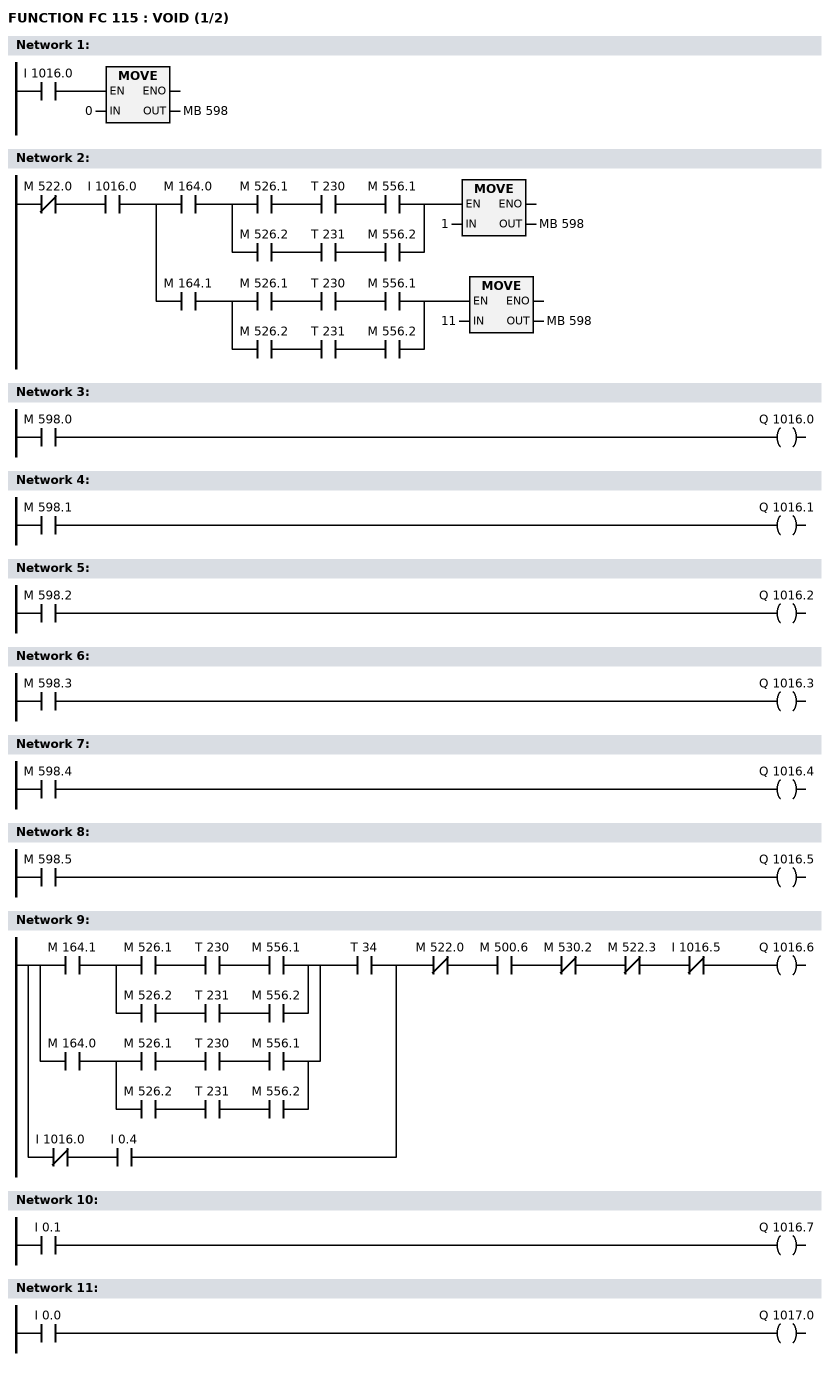

      A     I   1016.0;
      JNB   _001;
      L     0;
      T     MB   598;
_001: NOP   0;
NETWORK
TITLE =

      AN    M    522.0;
      A     I   1016.0;
      =     L      0.0;
      A     L      0.0;
      A     M    164.0;
      A(    ;
      A     M    526.1;
      A     T    230;
      A     M    556.1;
      O     ;
      A     M    526.2;
      A     T    231;
      A     M    556.2;
      )     ;
      JNB   _002;
      L     1;
      T     MB   598;
_002: NOP   0;
      A     L      0.0;
      A     M    164.1;
      A(    ;
      A     M    526.1;
      A     T    230;
      A     M    556.1;
      O     ;
      A     M    526.2;
      A     T    231;
      A     M    556.2;
      )     ;
      JNB   _003;
      L     11;
      T     MB   598;
_003: NOP   0;
NETWORK
TITLE =

      A     M    598.0;
      =     Q   1016.0;
NETWORK
TITLE =

      A     M    598.1;
      =     Q   1016.1;
NETWORK
TITLE =

      A     M    598.2;
      =     Q   1016.2;
NETWORK
TITLE =

      A     M    598.3;
      =     Q   1016.3;
NETWORK
TITLE =

      A     M    598.4;
      =     Q   1016.4;
NETWORK
TITLE =

      A     M    598.5;
      =     Q   1016.5;
NETWORK
TITLE =

      A(    ;
      A(    ;
      A     M    164.1;
      A(    ;
      A     M    526.1;
      A     T    230;
      A     M    556.1;
      O     ;
      A     M    526.2;
      A     T    231;
      A     M    556.2;
      )     ;
      O     ;
      A     M    164.0;
      A(    ;
      A     M    526.1;
      A     T    230;
      A     M    556.1;
      O     ;
      A     M    526.2;
      A     T    231;
      A     M    556.2;
      )     ;
      )     ;
      A     T     34;
      O     ;
      AN    I   1016.0;
      A     I      0.4;
      )     ;
      AN    M    522.0;
      A     M    500.6;
      AN    M    530.2;
      AN    M    522.3;
      AN    I   1016.5;
      =     Q   1016.6;
NETWORK
TITLE =

      A     I      0.1;
      =     Q   1016.7;
NETWORK
TITLE =

      A     I      0.0;
      =     Q   1017.0;
NETWORK
TITLE =
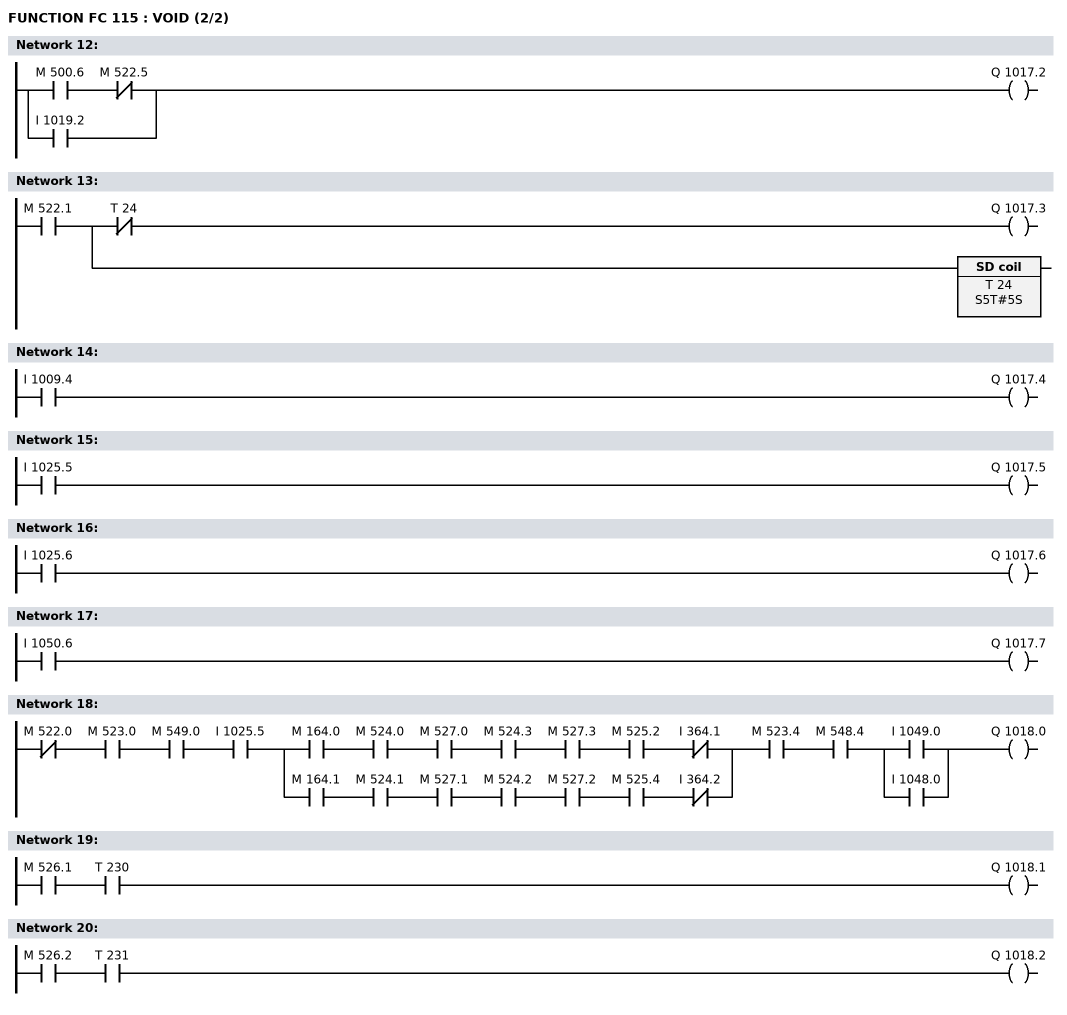

      A     M    500.6;
      AN    M    522.5;
      O     I   1019.2;
      =     Q   1017.2;
NETWORK
TITLE =

      A     M    522.1;
      =     L      0.0;
      A     L      0.0;
      AN    T     24;
      =     Q   1017.3;
      A     L      0.0;
      BLD   102;
      L     S5T#5S;
      SD    T     24;
NETWORK
TITLE =

      A     I   1009.4;
      =     Q   1017.4;
NETWORK
TITLE =

      A     I   1025.5;
      =     Q   1017.5;
NETWORK
TITLE =

      A     I   1025.6;
      =     Q   1017.6;
NETWORK
TITLE =

      A     I   1050.6;
      =     Q   1017.7;
NETWORK
TITLE =

      AN    M    522.0;
      A     M    523.0;
      A     M    549.0;
      A     I   1025.5;
      A(    ;
      A     M    164.0;
      A     M    524.0;
      A     M    527.0;
      A     M    524.3;
      A     M    527.3;
      A     M    525.2;
      AN    I    364.1;
      O     ;
      A     M    164.1;
      A     M    524.1;
      A     M    527.1;
      A     M    524.2;
      A     M    527.2;
      A     M    525.4;
      AN    I    364.2;
      )     ;
      A     M    523.4;
      A     M    548.4;
      A(    ;
      O     I   1049.0;
      O     I   1048.0;
      )     ;
      =     Q   1018.0;
NETWORK
TITLE =

      A     M    526.1;
      A     T    230;
      =     Q   1018.1;
NETWORK
TITLE =

      A     M    526.2;
      A     T    231;
      =     Q   1018.2;
END_FUNCTION

FUNCTION FC 116 : VOID
TITLE =
VERSION : 0.1

BEGIN
NETWORK
TITLE =
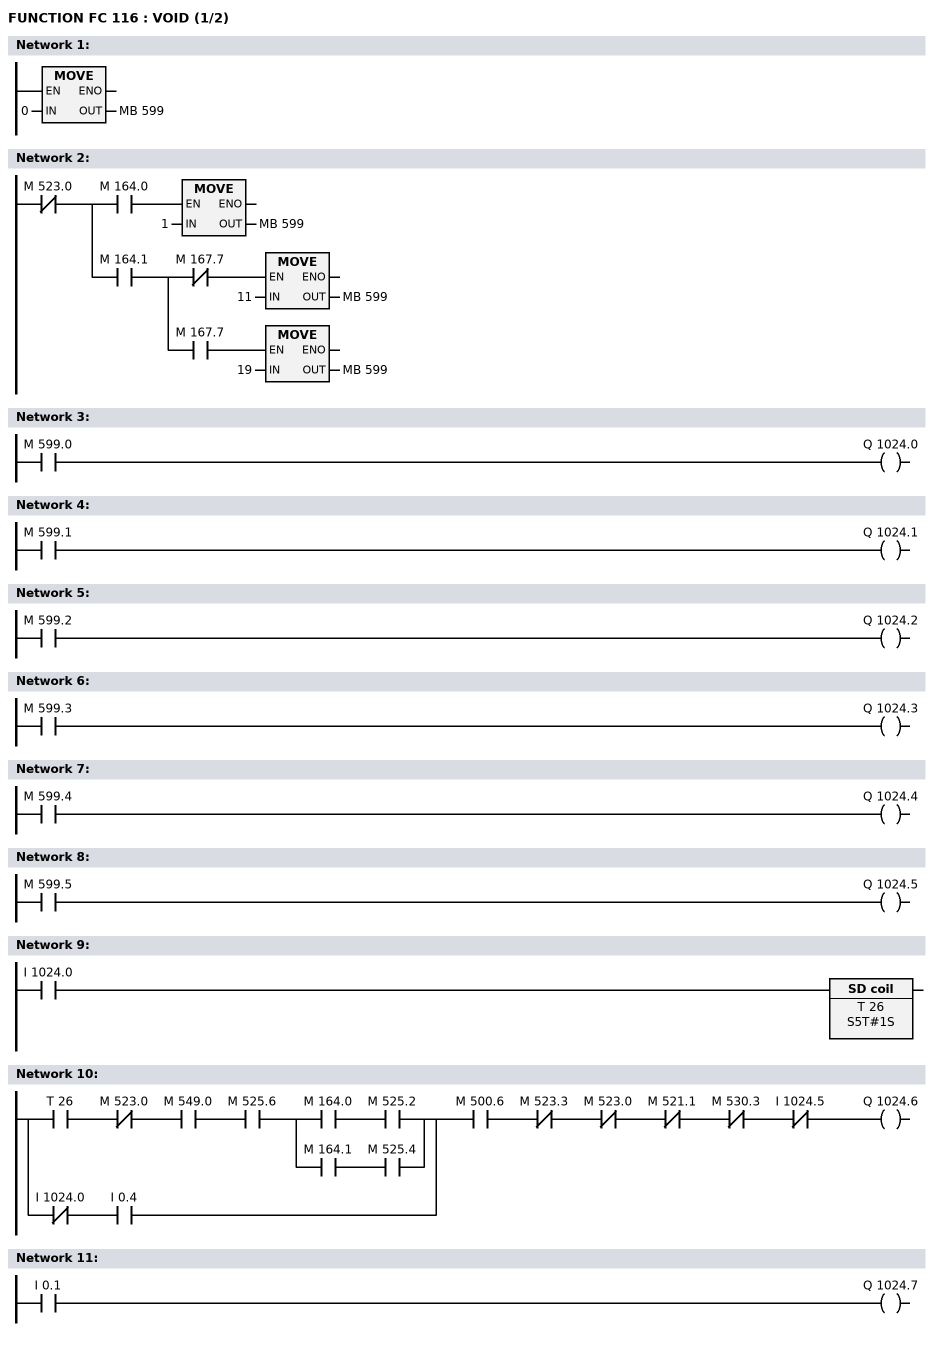

      L     0;
      T     MB   599;
      NOP   0;
NETWORK
TITLE =

      AN    M    523.0;
      =     L      0.0;
      A     L      0.0;
      A     M    164.0;
      JNB   _001;
      L     1;
      T     MB   599;
_001: NOP   0;
      A     L      0.0;
      A     M    164.1;
      =     L      0.1;
      A     L      0.1;
      AN    M    167.7;
      JNB   _002;
      L     11;
      T     MB   599;
_002: NOP   0;
      A     L      0.1;
      A     M    167.7;
      JNB   _003;
      L     19;
      T     MB   599;
_003: NOP   0;
NETWORK
TITLE =

      A     M    599.0;
      =     Q   1024.0;
NETWORK
TITLE =

      A     M    599.1;
      =     Q   1024.1;
NETWORK
TITLE =

      A     M    599.2;
      =     Q   1024.2;
NETWORK
TITLE =

      A     M    599.3;
      =     Q   1024.3;
NETWORK
TITLE =

      A     M    599.4;
      =     Q   1024.4;
NETWORK
TITLE =

      A     M    599.5;
      =     Q   1024.5;
NETWORK
TITLE =

      A     I   1024.0;
      L     S5T#1S;
      SD    T     26;
NETWORK
TITLE =

      A(    ;
      A     T     26;
      AN    M    523.0;
      A     M    549.0;
      A     M    525.6;
      A(    ;
      A     M    164.0;
      A     M    525.2;
      O     ;
      A     M    164.1;
      A     M    525.4;
      )     ;
      O     ;
      AN    I   1024.0;
      A     I      0.4;
      )     ;
      A     M    500.6;
      AN    M    523.3;
      AN    M    523.0;
      AN    M    521.1;
      AN    M    530.3;
      AN    I   1024.5;
      =     Q   1024.6;
NETWORK
TITLE =

      A     I      0.1;
      =     Q   1024.7;
NETWORK
TITLE =
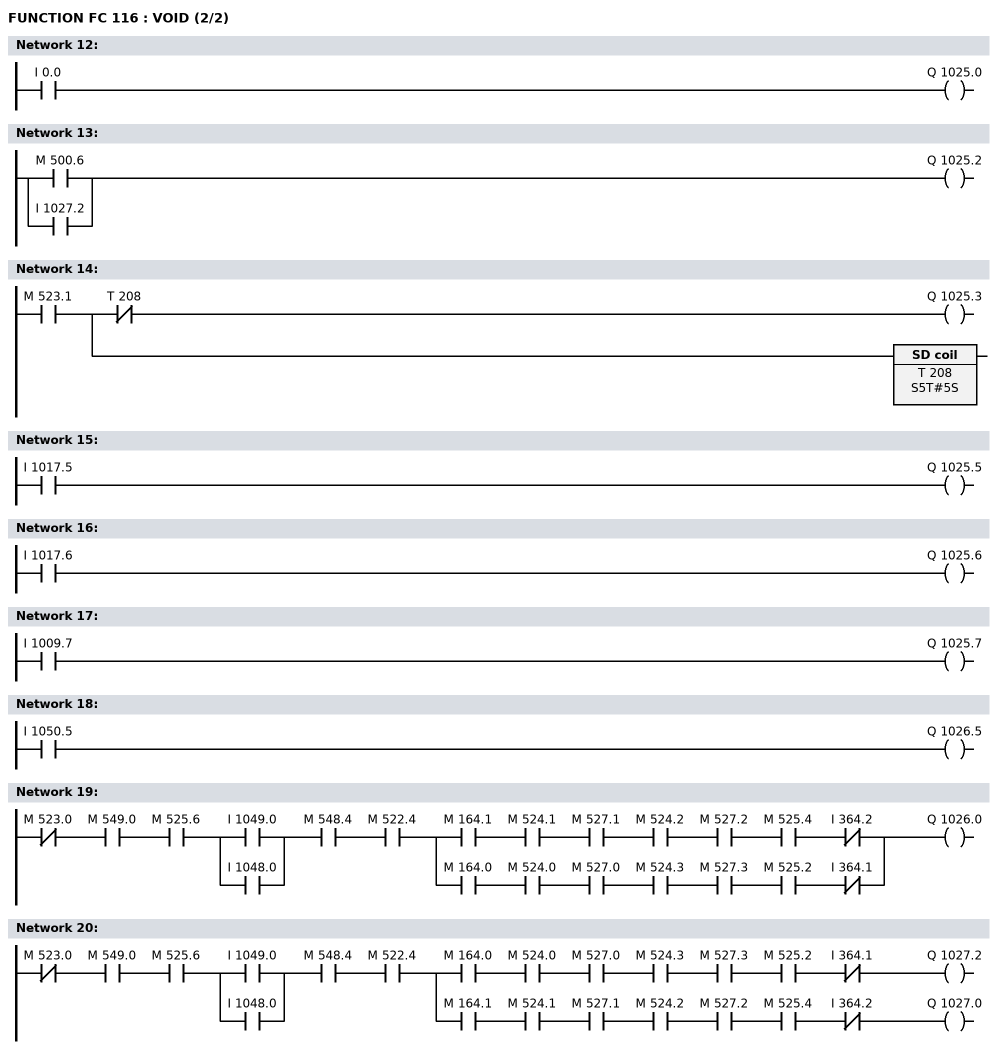

      A     I      0.0;
      =     Q   1025.0;
NETWORK
TITLE =

      O     M    500.6;
      O     I   1027.2;
      =     Q   1025.2;
NETWORK
TITLE =

      A     M    523.1;
      =     L      0.0;
      A     L      0.0;
      AN    T    208;
      =     Q   1025.3;
      A     L      0.0;
      BLD   102;
      L     S5T#5S;
      SD    T    208;
NETWORK
TITLE =

      A     I   1017.5;
      =     Q   1025.5;
NETWORK
TITLE =

      A     I   1017.6;
      =     Q   1025.6;
NETWORK
TITLE =

      A     I   1009.7;
      =     Q   1025.7;
NETWORK
TITLE =

      A     I   1050.5;
      =     Q   1026.5;
NETWORK
TITLE =

      AN    M    523.0;
      A     M    549.0;
      A     M    525.6;
      A(    ;
      O     I   1049.0;
      O     I   1048.0;
      )     ;
      A     M    548.4;
      A     M    522.4;
      A(    ;
      A     M    164.1;
      A     M    524.1;
      A     M    527.1;
      A     M    524.2;
      A     M    527.2;
      A     M    525.4;
      AN    I    364.2;
      O     ;
      A     M    164.0;
      A     M    524.0;
      A     M    527.0;
      A     M    524.3;
      A     M    527.3;
      A     M    525.2;
      AN    I    364.1;
      )     ;
      =     Q   1026.0;
NETWORK
TITLE =

      AN    M    523.0;
      A     M    549.0;
      A     M    525.6;
      A(    ;
      O     I   1049.0;
      O     I   1048.0;
      )     ;
      A     M    548.4;
      A     M    522.4;
      =     L      0.0;
      A     L      0.0;
      A     M    164.0;
      A     M    524.0;
      A     M    527.0;
      A     M    524.3;
      A     M    527.3;
      A     M    525.2;
      AN    I    364.1;
      =     Q   1027.2;
      A     L      0.0;
      A     M    164.1;
      A     M    524.1;
      A     M    527.1;
      A     M    524.2;
      A     M    527.2;
      A     M    525.4;
      AN    I    364.2;
      =     Q   1027.0;
END_FUNCTION

FUNCTION FC 117 : VOID
TITLE =
VERSION : 0.1

BEGIN
NETWORK
TITLE =

      AN    OV;
      L     S5T#3S;
      SD    T     59;
NETWORK
TITLE =

      AN    OV;
      =     L      0.0;
      A     L      0.0;
      A     M    500.5;
      A     DB49.DBX    2.0;
      S     M    571.0;
      A     L      0.0;
      AN    M    500.5;
      R     M    571.0;
      A     L      0.0;
      A     M    571.0;
      =     DB49.DBX    2.1;
NETWORK
TITLE =

      AN    OV;
      =     L      0.0;
      A     L      0.0;
      A(    ;
      A     T    323;
      A     DB49.DBX    2.1;
      A     DB49.DBX    3.0;
      O     ;
      A     M    573.0;
      A     M    573.1;
      O     ;
      AN    M    573.0;
      AN    M    573.1;
      )     ;
      S     M    573.0;
      R     M    573.1;
      A     L      0.0;
      A     T    323;
      A     DB49.DBX    2.1;
      A     DB49.DBX    3.1;
      S     M    573.1;
      R     M    573.0;
      A     L      0.0;
      A     M    573.0;
      =     DB49.DBX    3.2;
      A     L      0.0;
      A     M    573.1;
      =     DB49.DBX    3.3;
NETWORK
TITLE =

      AN    OV;
      =     L      0.0;
      A     L      0.0;
      A(    ;
      A     I     62.6;
      AN    I     62.7;
      O     ;
      AN    I     62.6;
      A     I     62.7;
      O     ;
      AN    I     62.6;
      AN    I     62.7;
      A     I     48.4;
      )     ;
      =     L      0.1;
      A     L      0.1;
      A     T    343;
      =     DB49.DBX    0.0;
      A     L      0.1;
      BLD   102;
      L     S5T#2S;
      SD    T    343;
      A     L      0.0;
      A(    ;
      A     DB49.DBX    3.2;
      A     I     62.4;
      O     ;
      A     DB49.DBX    3.3;
      AN    I     62.4;
      )     ;
      A     I     62.6;
      A     I     62.7;
      A     I     48.4;
      AN    T    323;
      =     L      0.1;
      A     L      0.1;
      A     T    413;
      =     DB49.DBX    1.0;
      A     L      0.1;
      BLD   102;
      L     S5T#3S;
      SD    T    413;
NETWORK
TITLE =
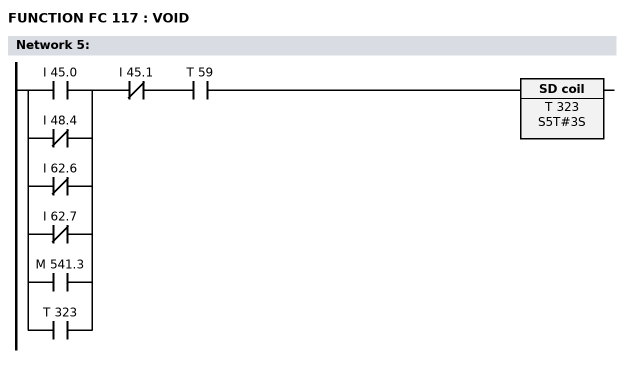

      A(    ;
      O     I     45.0;
      ON    I     48.4;
      ON    I     62.6;
      ON    I     62.7;
      O     M    541.3;
      O     T    323;
      )     ;
      AN    I     45.1;
      A     T     59;
      L     S5T#3S;
      SD    T    323;
NETWORK
TITLE =

      AN    OV;
      =     L      0.0;
      A     L      0.0;
      A     T    323;
      A     M      0.5;
      =     Q     53.0;
      A     L      0.0;
      AN    T    323;
      A(    ;
      O     T    303;
      O     T     63;
      )     ;
      =     Q     53.1;
      A     L      0.0;
      A     I     48.4;
      A     I     62.6;
      A     I     62.7;
      =     L      0.1;
      A     L      0.1;
      A     DB49.DBX    3.2;
      AN    DB49.DBX    3.3;
      =     L      0.2;
      A     L      0.2;
      BLD   102;
      L     S5T#3S;
      SD    T    303;
      A     L      0.2;
      A     T    303;
      =     DB49.DBX    3.4;
      A     L      0.1;
      A     DB49.DBX    3.3;
      AN    DB49.DBX    3.2;
      =     L      0.2;
      A     L      0.2;
      BLD   102;
      L     S5T#3S;
      SD    T     63;
      A     L      0.2;
      A     T     63;
      =     DB49.DBX    3.5;
NETWORK
TITLE =
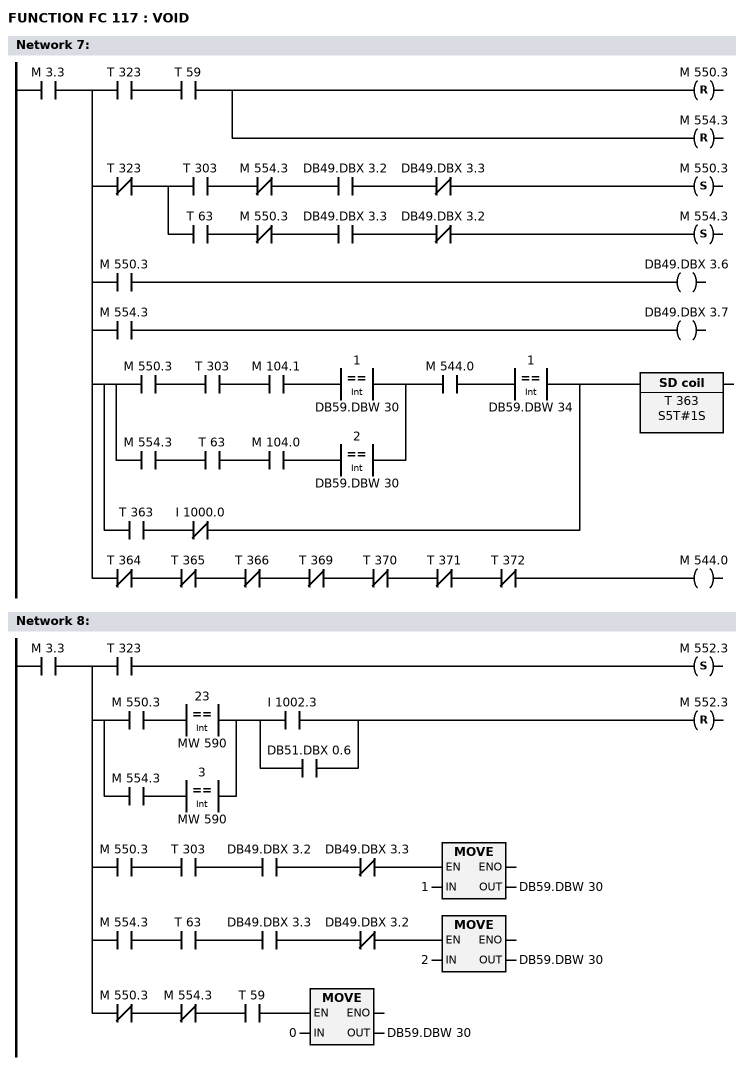

      A     M      3.3;
      =     L      0.0;
      A     L      0.0;
      A     T    323;
      A     T     59;
      R     M    550.3;
      R     M    554.3;
      A     L      0.0;
      AN    T    323;
      =     L      0.1;
      A     L      0.1;
      A     T    303;
      AN    M    554.3;
      A     DB49.DBX    3.2;
      AN    DB49.DBX    3.3;
      S     M    550.3;
      A     L      0.1;
      A     T     63;
      AN    M    550.3;
      A     DB49.DBX    3.3;
      AN    DB49.DBX    3.2;
      S     M    554.3;
      A     L      0.0;
      A     M    550.3;
      =     DB49.DBX    3.6;
      A     L      0.0;
      A     M    554.3;
      =     DB49.DBX    3.7;
      A     L      0.0;
      A(    ;
      A(    ;
      A     M    550.3;
      A     T    303;
      A     M    104.1;
      A(    ;
      L     1;
      L     DB59.DBW   30;
      ==I   ;
      )     ;
      O     ;
      A     M    554.3;
      A     T     63;
      A     M    104.0;
      A(    ;
      L     2;
      L     DB59.DBW   30;
      ==I   ;
      )     ;
      )     ;
      A     M    544.0;
      A(    ;
      L     1;
      L     DB59.DBW   34;
      ==I   ;
      )     ;
      O     ;
      A     T    363;
      AN    I   1000.0;
      )     ;
      L     S5T#1S;
      SD    T    363;
      A     L      0.0;
      AN    T    364;
      AN    T    365;
      AN    T    366;
      AN    T    369;
      AN    T    370;
      AN    T    371;
      AN    T    372;
      =     M    544.0;
NETWORK
TITLE =

      A     M      3.3;
      =     L      0.0;
      A     L      0.0;
      A     T    323;
      S     M    552.3;
      A     L      0.0;
      A(    ;
      A     M    550.3;
      A(    ;
      L     23;
      L     MW   590;
      ==I   ;
      )     ;
      O     ;
      A     M    554.3;
      A(    ;
      L     3;
      L     MW   590;
      ==I   ;
      )     ;
      )     ;
      A(    ;
      O     I   1002.3;
      O     DB51.DBX    0.6;
      )     ;
      R     M    552.3;
      A     L      0.0;
      A     M    550.3;
      A     T    303;
      A     DB49.DBX    3.2;
      AN    DB49.DBX    3.3;
      JNB   _001;
      L     1;
      T     DB59.DBW   30;
_001: NOP   0;
      A     L      0.0;
      A     M    554.3;
      A     T     63;
      A     DB49.DBX    3.3;
      AN    DB49.DBX    3.2;
      JNB   _002;
      L     2;
      T     DB59.DBW   30;
_002: NOP   0;
      A     L      0.0;
      AN    M    550.3;
      AN    M    554.3;
      A     T     59;
      JNB   _003;
      L     0;
      T     DB59.DBW   30;
_003: NOP   0;
NETWORK
TITLE =

      AN    OV;
      =     L      0.0;
      A     L      0.0;
      A(    ;
      A     T    324;
      A     DB49.DBX    2.1;
      A     DB49.DBX    4.0;
      O     ;
      A     M    574.0;
      A     M    574.1;
      O     ;
      AN    M    574.0;
      AN    M    574.1;
      )     ;
      S     M    574.0;
      R     M    574.1;
      A     L      0.0;
      A     T    324;
      A     DB49.DBX    2.1;
      A     DB49.DBX    4.1;
      S     M    574.1;
      R     M    574.0;
      A     L      0.0;
      A     M    574.0;
      =     DB49.DBX    4.2;
      A     L      0.0;
      A     M    574.1;
      =     DB49.DBX    4.3;
NETWORK
TITLE =

      AN    OV;
      =     L      0.0;
      A     L      0.0;
      A(    ;
      A     I     63.4;
      AN    I     63.5;
      O     ;
      AN    I     63.4;
      A     I     63.5;
      O     ;
      AN    I     63.4;
      AN    I     63.5;
      A     I     48.1;
      )     ;
      =     L      0.1;
      A     L      0.1;
      A     T    344;
      =     DB49.DBX    0.1;
      A     L      0.1;
      BLD   102;
      L     S5T#2S;
      SD    T    344;
      A     L      0.0;
      A(    ;
      A     DB49.DBX    4.2;
      A     I     62.5;
      O     ;
      A     DB49.DBX    4.3;
      AN    I     62.5;
      )     ;
      A     I     63.4;
      A     I     63.5;
      A     I     48.1;
      AN    T    324;
      =     L      0.1;
      A     L      0.1;
      A     T    414;
      =     DB49.DBX    1.1;
      A     L      0.1;
      BLD   102;
      L     S5T#3S;
      SD    T    414;
NETWORK
TITLE =
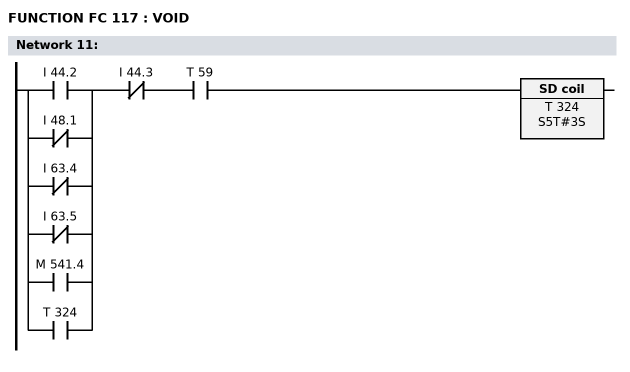

      A(    ;
      O     I     44.2;
      ON    I     48.1;
      ON    I     63.4;
      ON    I     63.5;
      O     M    541.4;
      O     T    324;
      )     ;
      AN    I     44.3;
      A     T     59;
      L     S5T#3S;
      SD    T    324;
NETWORK
TITLE =

      AN    OV;
      =     L      0.0;
      A     L      0.0;
      A     T    324;
      A     M      0.5;
      =     Q     52.2;
      A     L      0.0;
      AN    T    324;
      A(    ;
      O     T    304;
      O     T     64;
      )     ;
      =     Q     52.3;
      A     L      0.0;
      A     I     48.1;
      A     I     63.4;
      A     I     63.5;
      =     L      0.1;
      A     L      0.1;
      A     DB49.DBX    4.2;
      AN    DB49.DBX    4.3;
      =     L      0.2;
      A     L      0.2;
      BLD   102;
      L     S5T#3S;
      SD    T    304;
      A     L      0.2;
      A     T    304;
      =     DB49.DBX    4.4;
      A     L      0.1;
      A     DB49.DBX    4.3;
      AN    DB49.DBX    4.2;
      =     L      0.2;
      A     L      0.2;
      BLD   102;
      L     S5T#3S;
      SD    T     64;
      A     L      0.2;
      A     T     64;
      =     DB49.DBX    4.5;
NETWORK
TITLE =
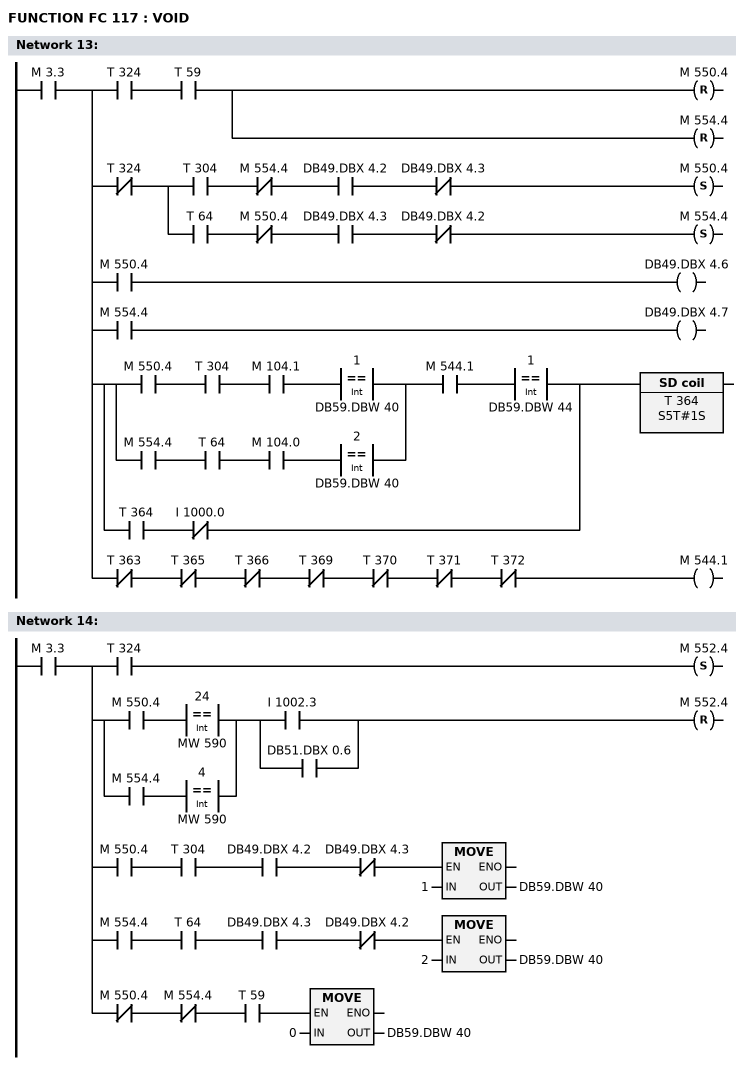

      A     M      3.3;
      =     L      0.0;
      A     L      0.0;
      A     T    324;
      A     T     59;
      R     M    550.4;
      R     M    554.4;
      A     L      0.0;
      AN    T    324;
      =     L      0.1;
      A     L      0.1;
      A     T    304;
      AN    M    554.4;
      A     DB49.DBX    4.2;
      AN    DB49.DBX    4.3;
      S     M    550.4;
      A     L      0.1;
      A     T     64;
      AN    M    550.4;
      A     DB49.DBX    4.3;
      AN    DB49.DBX    4.2;
      S     M    554.4;
      A     L      0.0;
      A     M    550.4;
      =     DB49.DBX    4.6;
      A     L      0.0;
      A     M    554.4;
      =     DB49.DBX    4.7;
      A     L      0.0;
      A(    ;
      A(    ;
      A     M    550.4;
      A     T    304;
      A     M    104.1;
      A(    ;
      L     1;
      L     DB59.DBW   40;
      ==I   ;
      )     ;
      O     ;
      A     M    554.4;
      A     T     64;
      A     M    104.0;
      A(    ;
      L     2;
      L     DB59.DBW   40;
      ==I   ;
      )     ;
      )     ;
      A     M    544.1;
      A(    ;
      L     1;
      L     DB59.DBW   44;
      ==I   ;
      )     ;
      O     ;
      A     T    364;
      AN    I   1000.0;
      )     ;
      L     S5T#1S;
      SD    T    364;
      A     L      0.0;
      AN    T    363;
      AN    T    365;
      AN    T    366;
      AN    T    369;
      AN    T    370;
      AN    T    371;
      AN    T    372;
      =     M    544.1;
NETWORK
TITLE =

      A     M      3.3;
      =     L      0.0;
      A     L      0.0;
      A     T    324;
      S     M    552.4;
      A     L      0.0;
      A(    ;
      A     M    550.4;
      A(    ;
      L     24;
      L     MW   590;
      ==I   ;
      )     ;
      O     ;
      A     M    554.4;
      A(    ;
      L     4;
      L     MW   590;
      ==I   ;
      )     ;
      )     ;
      A(    ;
      O     I   1002.3;
      O     DB51.DBX    0.6;
      )     ;
      R     M    552.4;
      A     L      0.0;
      A     M    550.4;
      A     T    304;
      A     DB49.DBX    4.2;
      AN    DB49.DBX    4.3;
      JNB   _004;
      L     1;
      T     DB59.DBW   40;
_004: NOP   0;
      A     L      0.0;
      A     M    554.4;
      A     T     64;
      A     DB49.DBX    4.3;
      AN    DB49.DBX    4.2;
      JNB   _005;
      L     2;
      T     DB59.DBW   40;
_005: NOP   0;
      A     L      0.0;
      AN    M    550.4;
      AN    M    554.4;
      A     T     59;
      JNB   _006;
      L     0;
      T     DB59.DBW   40;
_006: NOP   0;
NETWORK
TITLE =

      AN    OV;
      =     L      0.0;
      A     L      0.0;
      A(    ;
      A     T    325;
      A     DB49.DBX    2.1;
      A     DB49.DBX    5.0;
      O     ;
      A     M    575.0;
      A     M    575.1;
      O     ;
      AN    M    575.0;
      AN    M    575.1;
      )     ;
      S     M    575.0;
      R     M    575.1;
      A     L      0.0;
      A     T    325;
      A     DB49.DBX    2.1;
      A     DB49.DBX    5.1;
      S     M    575.1;
      R     M    575.0;
      A     L      0.0;
      A     M    575.0;
      =     DB49.DBX    5.2;
      A     L      0.0;
      A     M    575.1;
      =     DB49.DBX    5.3;
NETWORK
TITLE =

      AN    OV;
      =     L      0.0;
      A     L      0.0;
      A(    ;
      A     I     63.0;
      AN    I     63.1;
      O     ;
      AN    I     63.0;
      A     I     63.1;
      O     ;
      AN    I     63.0;
      AN    I     63.1;
      A     I     48.5;
      )     ;
      =     L      0.1;
      A     L      0.1;
      A     T    345;
      =     DB49.DBX    0.2;
      A     L      0.1;
      BLD   102;
      L     S5T#2S;
      SD    T    345;
      A     L      0.0;
      A(    ;
      A     DB49.DBX    5.2;
      A     I     63.2;
      O     ;
      A     DB49.DBX    5.3;
      AN    I     63.2;
      )     ;
      A     I     63.0;
      A     I     63.1;
      A     I     48.5;
      AN    T    325;
      =     L      0.1;
      A     L      0.1;
      A     T    415;
      =     DB49.DBX    1.2;
      A     L      0.1;
      BLD   102;
      L     S5T#3S;
      SD    T    415;
NETWORK
TITLE =
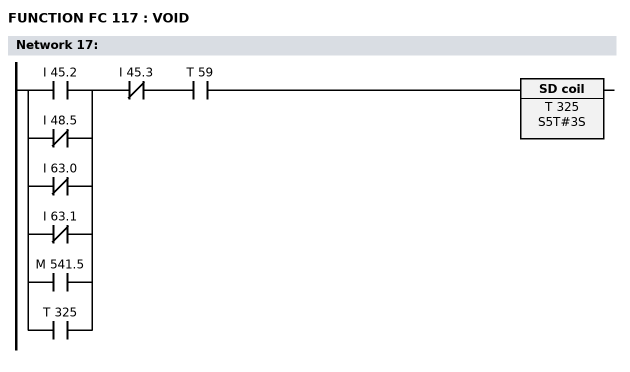

      A(    ;
      O     I     45.2;
      ON    I     48.5;
      ON    I     63.0;
      ON    I     63.1;
      O     M    541.5;
      O     T    325;
      )     ;
      AN    I     45.3;
      A     T     59;
      L     S5T#3S;
      SD    T    325;
NETWORK
TITLE =

      AN    OV;
      =     L      0.0;
      A     L      0.0;
      A     T    325;
      A     M      0.5;
      =     Q     53.2;
      A     L      0.0;
      AN    T    325;
      A(    ;
      O     T    305;
      O     T     65;
      )     ;
      =     Q     53.3;
      A     L      0.0;
      A     I     48.5;
      A     I     63.0;
      A     I     63.1;
      =     L      0.1;
      A     L      0.1;
      A     DB49.DBX    5.2;
      AN    DB49.DBX    5.3;
      =     L      0.2;
      A     L      0.2;
      BLD   102;
      L     S5T#3S;
      SD    T    305;
      A     L      0.2;
      A     T    305;
      =     DB49.DBX    5.4;
      A     L      0.1;
      A     DB49.DBX    5.3;
      AN    DB49.DBX    5.2;
      =     L      0.2;
      A     L      0.2;
      BLD   102;
      L     S5T#3S;
      SD    T     65;
      A     L      0.2;
      A     T     65;
      =     DB49.DBX    5.5;
NETWORK
TITLE =
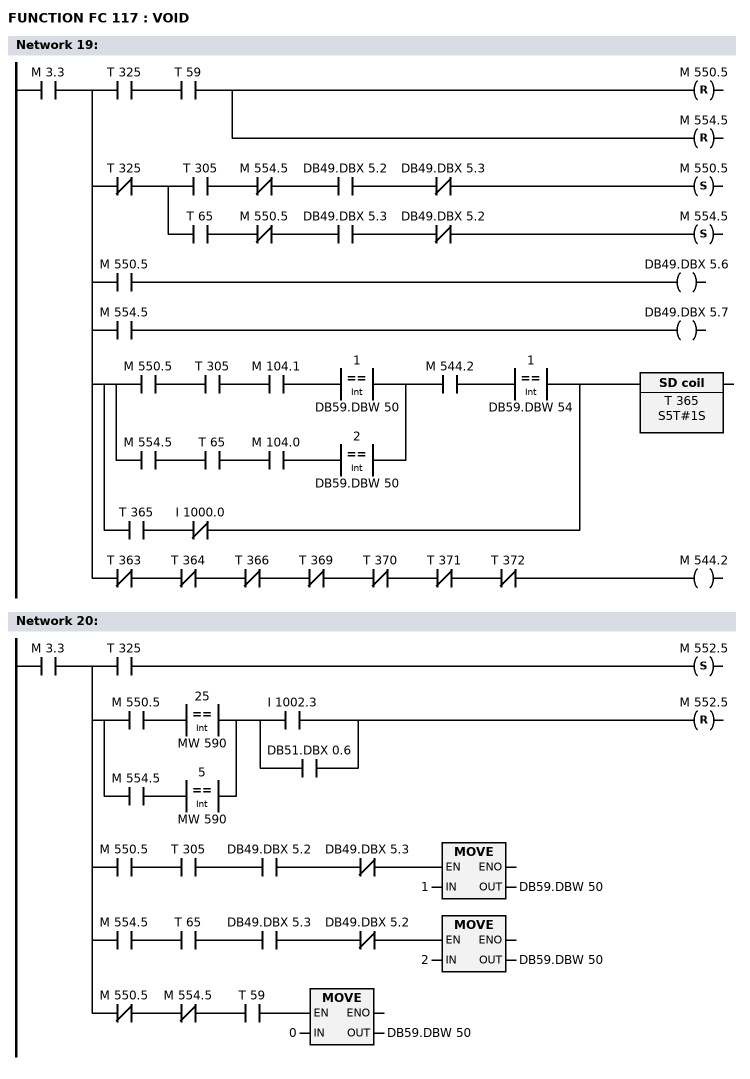

      A     M      3.3;
      =     L      0.0;
      A     L      0.0;
      A     T    325;
      A     T     59;
      R     M    550.5;
      R     M    554.5;
      A     L      0.0;
      AN    T    325;
      =     L      0.1;
      A     L      0.1;
      A     T    305;
      AN    M    554.5;
      A     DB49.DBX    5.2;
      AN    DB49.DBX    5.3;
      S     M    550.5;
      A     L      0.1;
      A     T     65;
      AN    M    550.5;
      A     DB49.DBX    5.3;
      AN    DB49.DBX    5.2;
      S     M    554.5;
      A     L      0.0;
      A     M    550.5;
      =     DB49.DBX    5.6;
      A     L      0.0;
      A     M    554.5;
      =     DB49.DBX    5.7;
      A     L      0.0;
      A(    ;
      A(    ;
      A     M    550.5;
      A     T    305;
      A     M    104.1;
      A(    ;
      L     1;
      L     DB59.DBW   50;
      ==I   ;
      )     ;
      O     ;
      A     M    554.5;
      A     T     65;
      A     M    104.0;
      A(    ;
      L     2;
      L     DB59.DBW   50;
      ==I   ;
      )     ;
      )     ;
      A     M    544.2;
      A(    ;
      L     1;
      L     DB59.DBW   54;
      ==I   ;
      )     ;
      O     ;
      A     T    365;
      AN    I   1000.0;
      )     ;
      L     S5T#1S;
      SD    T    365;
      A     L      0.0;
      AN    T    363;
      AN    T    364;
      AN    T    366;
      AN    T    369;
      AN    T    370;
      AN    T    371;
      AN    T    372;
      =     M    544.2;
NETWORK
TITLE =

      A     M      3.3;
      =     L      0.0;
      A     L      0.0;
      A     T    325;
      S     M    552.5;
      A     L      0.0;
      A(    ;
      A     M    550.5;
      A(    ;
      L     25;
      L     MW   590;
      ==I   ;
      )     ;
      O     ;
      A     M    554.5;
      A(    ;
      L     5;
      L     MW   590;
      ==I   ;
      )     ;
      )     ;
      A(    ;
      O     I   1002.3;
      O     DB51.DBX    0.6;
      )     ;
      R     M    552.5;
      A     L      0.0;
      A     M    550.5;
      A     T    305;
      A     DB49.DBX    5.2;
      AN    DB49.DBX    5.3;
      JNB   _007;
      L     1;
      T     DB59.DBW   50;
_007: NOP   0;
      A     L      0.0;
      A     M    554.5;
      A     T     65;
      A     DB49.DBX    5.3;
      AN    DB49.DBX    5.2;
      JNB   _008;
      L     2;
      T     DB59.DBW   50;
_008: NOP   0;
      A     L      0.0;
      AN    M    550.5;
      AN    M    554.5;
      A     T     59;
      JNB   _009;
      L     0;
      T     DB59.DBW   50;
_009: NOP   0;
NETWORK
TITLE =

      AN    OV;
      =     L      0.0;
      A     L      0.0;
      A(    ;
      A     T    326;
      A     DB49.DBX    2.1;
      A     DB49.DBX    6.0;
      O     ;
      A     M    576.0;
      A     M    576.1;
      O     ;
      AN    M    576.0;
      AN    M    576.1;
      )     ;
      S     M    576.0;
      R     M    576.1;
      A     L      0.0;
      A     T    326;
      A     DB49.DBX    2.1;
      A     DB49.DBX    6.1;
      S     M    576.1;
      R     M    576.0;
      A     L      0.0;
      A     M    576.0;
      =     DB49.DBX    6.2;
      A     L      0.0;
      A     M    576.1;
      =     DB49.DBX    6.3;
NETWORK
TITLE =

      AN    OV;
      =     L      0.0;
      A     L      0.0;
      A(    ;
      A     I     63.6;
      AN    I     63.7;
      O     ;
      AN    I     63.6;
      A     I     63.7;
      O     ;
      AN    I     63.6;
      AN    I     63.7;
      A     I     48.2;
      )     ;
      =     L      0.1;
      A     L      0.1;
      A     T    346;
      =     DB49.DBX    0.3;
      A     L      0.1;
      BLD   102;
      L     S5T#2S;
      SD    T    346;
      A     L      0.0;
      A(    ;
      A     DB49.DBX    6.2;
      A     I     63.3;
      O     ;
      A     DB49.DBX    6.3;
      AN    I     63.3;
      )     ;
      A     I     63.6;
      A     I     63.7;
      A     I     48.2;
      AN    T    326;
      =     L      0.1;
      A     L      0.1;
      A     T    416;
      =     DB49.DBX    1.3;
      A     L      0.1;
      BLD   102;
      L     S5T#3S;
      SD    T    416;
NETWORK
TITLE =
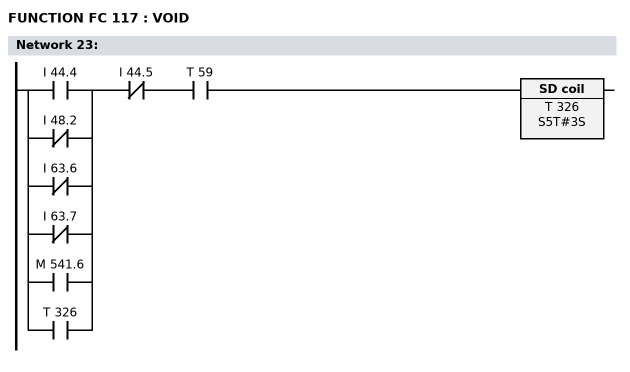

      A(    ;
      O     I     44.4;
      ON    I     48.2;
      ON    I     63.6;
      ON    I     63.7;
      O     M    541.6;
      O     T    326;
      )     ;
      AN    I     44.5;
      A     T     59;
      L     S5T#3S;
      SD    T    326;
NETWORK
TITLE =

      AN    OV;
      =     L      0.0;
      A     L      0.0;
      A     T    326;
      A     M      0.5;
      =     Q     52.4;
      A     L      0.0;
      AN    T    326;
      A(    ;
      O     T    306;
      O     T     66;
      )     ;
      =     Q     52.5;
      A     L      0.0;
      A     I     48.2;
      A     I     63.6;
      A     I     63.7;
      =     L      0.1;
      A     L      0.1;
      A     DB49.DBX    6.2;
      AN    DB49.DBX    6.3;
      =     L      0.2;
      A     L      0.2;
      BLD   102;
      L     S5T#3S;
      SD    T    306;
      A     L      0.2;
      A     T    306;
      =     DB49.DBX    6.4;
      A     L      0.1;
      A     DB49.DBX    6.3;
      AN    DB49.DBX    6.2;
      =     L      0.2;
      A     L      0.2;
      BLD   102;
      L     S5T#3S;
      SD    T     66;
      A     L      0.2;
      A     T     66;
      =     DB49.DBX    6.5;
NETWORK
TITLE =
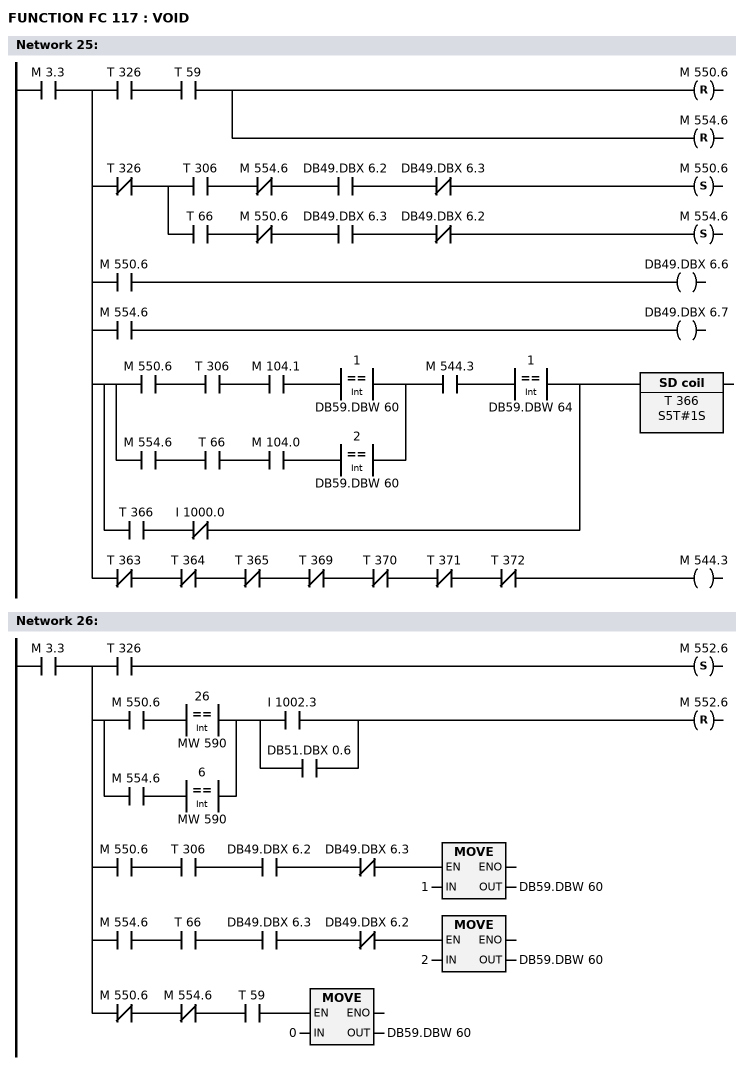

      A     M      3.3;
      =     L      0.0;
      A     L      0.0;
      A     T    326;
      A     T     59;
      R     M    550.6;
      R     M    554.6;
      A     L      0.0;
      AN    T    326;
      =     L      0.1;
      A     L      0.1;
      A     T    306;
      AN    M    554.6;
      A     DB49.DBX    6.2;
      AN    DB49.DBX    6.3;
      S     M    550.6;
      A     L      0.1;
      A     T     66;
      AN    M    550.6;
      A     DB49.DBX    6.3;
      AN    DB49.DBX    6.2;
      S     M    554.6;
      A     L      0.0;
      A     M    550.6;
      =     DB49.DBX    6.6;
      A     L      0.0;
      A     M    554.6;
      =     DB49.DBX    6.7;
      A     L      0.0;
      A(    ;
      A(    ;
      A     M    550.6;
      A     T    306;
      A     M    104.1;
      A(    ;
      L     1;
      L     DB59.DBW   60;
      ==I   ;
      )     ;
      O     ;
      A     M    554.6;
      A     T     66;
      A     M    104.0;
      A(    ;
      L     2;
      L     DB59.DBW   60;
      ==I   ;
      )     ;
      )     ;
      A     M    544.3;
      A(    ;
      L     1;
      L     DB59.DBW   64;
      ==I   ;
      )     ;
      O     ;
      A     T    366;
      AN    I   1000.0;
      )     ;
      L     S5T#1S;
      SD    T    366;
      A     L      0.0;
      AN    T    363;
      AN    T    364;
      AN    T    365;
      AN    T    369;
      AN    T    370;
      AN    T    371;
      AN    T    372;
      =     M    544.3;
NETWORK
TITLE =

      A     M      3.3;
      =     L      0.0;
      A     L      0.0;
      A     T    326;
      S     M    552.6;
      A     L      0.0;
      A(    ;
      A     M    550.6;
      A(    ;
      L     26;
      L     MW   590;
      ==I   ;
      )     ;
      O     ;
      A     M    554.6;
      A(    ;
      L     6;
      L     MW   590;
      ==I   ;
      )     ;
      )     ;
      A(    ;
      O     I   1002.3;
      O     DB51.DBX    0.6;
      )     ;
      R     M    552.6;
      A     L      0.0;
      A     M    550.6;
      A     T    306;
      A     DB49.DBX    6.2;
      AN    DB49.DBX    6.3;
      JNB   _00a;
      L     1;
      T     DB59.DBW   60;
_00a: NOP   0;
      A     L      0.0;
      A     M    554.6;
      A     T     66;
      A     DB49.DBX    6.3;
      AN    DB49.DBX    6.2;
      JNB   _00b;
      L     2;
      T     DB59.DBW   60;
_00b: NOP   0;
      A     L      0.0;
      AN    M    550.6;
      AN    M    554.6;
      A     T     59;
      JNB   _00c;
      L     0;
      T     DB59.DBW   60;
_00c: NOP   0;
NETWORK
TITLE =

      AN    OV;
      =     L      0.0;
      A     L      0.0;
      A(    ;
      A     T    329;
      A     DB49.DBX    2.1;
      A     DB49.DBX    9.0;
      O     ;
      A     M    579.0;
      A     M    579.1;
      O     ;
      AN    M    579.0;
      AN    M    579.1;
      )     ;
      S     M    579.0;
      R     M    579.1;
      A     L      0.0;
      A     T    329;
      A     DB49.DBX    2.1;
      A     DB49.DBX    9.1;
      S     M    579.1;
      R     M    579.0;
      A     L      0.0;
      A     M    579.0;
      =     DB49.DBX    9.2;
      A     L      0.0;
      A     M    579.1;
      =     DB49.DBX    9.3;
NETWORK
TITLE =

      AN    OV;
      =     L      0.0;
      A     L      0.0;
      A(    ;
      A     I     61.2;
      AN    I     61.3;
      O     ;
      AN    I     61.2;
      A     I     61.3;
      O     ;
      AN    I     61.2;
      AN    I     61.3;
      A     I     48.7;
      )     ;
      =     L      0.1;
      A     L      0.1;
      A     T    349;
      =     DB49.DBX    0.4;
      A     L      0.1;
      BLD   102;
      L     S5T#2S;
      SD    T    349;
      A     L      0.0;
      A(    ;
      A     DB49.DBX    9.2;
      A     I     61.0;
      O     ;
      A     DB49.DBX    9.3;
      AN    I     61.0;
      )     ;
      A     I     61.2;
      A     I     61.3;
      A     I     48.7;
      AN    T    329;
      =     L      0.1;
      A     L      0.1;
      A     T    419;
      =     DB49.DBX    1.4;
      A     L      0.1;
      BLD   102;
      L     S5T#3S;
      SD    T    419;
NETWORK
TITLE =
